{attribute 'Tc2GvlVarNames'}
VAR_GLOBAL

(* xxxxxxxxxxxxxxxxxxxxxxxxxxxxxxxx OUTPUT DWORD LINK with %MX10000-MX19000  xxxxxxxxxxxxxxxxxxxxxxxxxxxxxxxx*)
(*========================================================================*)

	WY10000 :DWORD; (* %MD10000 - GENERAL ALARM RESET IND (-100S1) *)
	WY10001 :DWORD; (* %MD10004 - GENERAL BUZZER RESET IND (-100S2) *)
	WY10002 :DWORD; (* %MD10008 - GENERAL BUZZER TONE 1 (-150H3) *)
	WY10003 :DWORD; (* %MD10012 - GENERAL BUZZER TONE 2 (-150H3) *)
	WY10004 :DWORD; (* %MD10016 - GENERAL TOWER LIGHT IND - RED (-150H5) *)
	WY10005 :DWORD; (* %MD10020 - GENERAL TOWER LIGHT IND - YELLOW (-150H5) *)
	WY10006 :DWORD; (* %MD10024 - GENERAL TOWER LIGHT IND - GREEN (-150H5) *)
	WY10007 :DWORD; (* %MD10028 - RESERVED *)
	WY10008 :DWORD; (* %MD10032 - RESERVED *)
	WY10009 :DWORD; (* %MD10036 - RESERVED *)
	WY10010 :DWORD; (* %MD10040 - RESERVED *)
	WY10011 :DWORD; (* %MD10044 - RESERVED *)
	WY10012 :DWORD; (* %MD10048 - RESERVED *)
	WY10013 :DWORD; (* %MD10052 - RESERVED *)
	WY10014 :DWORD; (* %MD10056 - RESERVED *)
	WY10015 :DWORD; (* %MD10060 - RESERVED *)

	WY10100 :DWORD; (* %MD10100 - STN 1 PROCESS TANK PUMP ON/OFF (-50K1) *)
	WY10101 :DWORD; (* %MD10104 - STN 2 PROCESS TANK PUMP ON/OFF (-51K1) *)
	WY10102 :DWORD; (* %MD10108 - STN 3 PROCESS TANK PUMP ON/OFF (-52K1) *)
	WY10103 :DWORD; (* %MD10112 - STN 5 VACUUM PUMP ON/OFF (-56K1) *)
	WY10104 :DWORD; (* %MD10116 - STN 2&3 AGITATION MOTOR ON/OFF (-25K1) *)
	WY10105 :DWORD; (* %MD10120 - STN 5 BLOWER ON/OFF (-65K1) *)
	WY10106 :DWORD; (* %MD10124 - STN 1 SUB PROCESS TANK STIRRING MOTOR ON/OFF (-26K1) *)
	WY10107 :DWORD; (* %MD10128 - DETERGENT TANK 1 STIRRING MOTOR ON/OFF (-27K1) *)
	WY10108 :DWORD; (* %MD10132 - STN 1 ULTRASONIC ON/OFF (-16K1) *)
	WY10109 :DWORD; (* %MD10136 - STN 2 ULTRASONIC ON/OFF (-17K1) *)
	WY10110 :DWORD; (* %MD10140 - STN 3 ULTRASONIC ON/OFF (-18K1) *)
	WY10111 :DWORD; (* %MD10144 - STN 1 ELECTRIC ACTUATOR ON/OFF (-21K1) *)
	WY10112 :DWORD; (* %MD10148 - STN 2 ELECTRIC ACTUATOR ON/OFF (-22K1) *)
	WY10113 :DWORD; (* %MD10152 - STN 3 ELECTRIC ACTUATOR ON/OFF (-23K1) *)
	WY10114 :DWORD; (* %MD10156 - RESERVED *)
	WY10115 :DWORD; (* %MD10160 - RESERVED *)

	WY10200 :DWORD; (* %MD10200 - STN 5 PROCESS TANK HEATER A ON/OFF (-70K1) *)
	WY10201 :DWORD; (* %MD10204 - STN 5 PROCESS TANK HEATER B ON/OFF (-71K1) *)
	WY10202 :DWORD; (* %MD10208 - STN 1 SUB PROCESS TANK HEATER ON/OFF (-72K1) *)
	WY10203 :DWORD; (* %MD10212 - STN 2 SUB PROCESS TANK HEATER ON/OFF (-73K1) *)
	WY10204 :DWORD; (* %MD10216 - STN 3 SUB PROCESS TANK HEATER ON/OFF (-74K1) *)
	WY10205 :DWORD; (* %MD10220 - MAIN INC HEATER ON/OFF   (-75K1) *)
	WY10206 :DWORD; (* %MD10224 - STN 1 ULTRASONIC FREQ ON/OFF (-16U1) *)
	WY10207 :DWORD; (* %MD10228 - STN 2 ULTRASONIC FREQ ON/OFF (-17U1) *)
	WY10208 :DWORD; (* %MD10232 - STN 3 ULTRASONIC FREQ ON/OFF (-18U1) *)
	WY10209 :DWORD; (* %MD10236 - RESERVED *)
	WY10210 :DWORD; (* %MD10240 - RESERVED *)
	WY10211 :DWORD; (* %MD10244 - RESERVED *)
	WY10212 :DWORD; (* %MD10248 - RESERVED *)
	WY10213 :DWORD; (* %MD10252 - RESERVED *)
	WY10214 :DWORD; (* %MD10256 - RESERVED *)
	WY10215 :DWORD; (* %MD10260 - RESERVED *)

	WY11500 :DWORD; (* %MD11500 - STN 1 SLIDING DOOR - OPEN (-160Y1) *)
	WY11501 :DWORD; (* %MD11504 - STN 1 SLIDING DOOR - CLOSE (-160Y2) *)
	WY11502 :DWORD; (* %MD11508 - STN 4 SLIDING DOOR - OPEN (-160Y3) *)
	WY11503 :DWORD; (* %MD11512 - STN 4 SLIDING DOOR - CLOSE (-160Y4) *)
	WY11504 :DWORD; (* %MD11516 - STN 5 SLIDING DOOR - OPEN (-160Y5) *)
	WY11505 :DWORD; (* %MD11520 - STN 5 SLIDING DOOR - CLOSE (-160Y6) *)
	WY11506 :DWORD; (* %MD11524 - STN 5 SLIDING DOOR - CLAMP (-160Y7) *)
	WY11507 :DWORD; (* %MD11528 - STN 5 SLIDING DOOR - UNCLAMP (-160Y8) *)
	WY11508 :DWORD; (* %MD11532 - LD CYLINDER - UP (-160Y9) *)
	WY11509 :DWORD; (* %MD11536 - LD CYLINDER - DOWN (-160Y10) *)
	WY11510 :DWORD; (* %MD11540 - LD CYLINDER - FRONT (-160Y11) *)
	WY11511 :DWORD; (* %MD11544 - LD CYLINDER - BACK (-160Y12) *)
	WY11512 :DWORD; (* %MD11548 - ULD CYLINDER - UP (-160Y13) *)
	WY11513 :DWORD; (* %MD11552 - ULD CYLINDER - DOWN (-160Y14) *)
	WY11514 :DWORD; (* %MD11556 - ULD CYLINDER - FRONT (-160Y15) *)
	WY11515 :DWORD; (* %MD11560 - ULD CYLINDER - BACK (-160Y16) *)

	WY11600 :DWORD; (* %MD11600 - GENERAL INCOMING DIW SUPPLY AVINC-1 (-161Y1) *)
	WY11601 :DWORD; (* %MD11604 - STN 1 PROCESS TANK INCOMING DI SUPPLY AV1-1 (-161Y2) *)
	WY11602 :DWORD; (* %MD11608 - STN 1 SUB TANK INCOMING DIW SUPPLY AV1-2 (-161Y3) *)
	WY11603 :DWORD; (* %MD11612 - STN 1 DETERGENT SUPPLY 3-2 WAY AV1-3 (-161Y4) *)
	WY11604 :DWORD; (* %MD11616 - STN 2 PROCESS TANK INCOMING DIW SUPPLY AV2-1 (-161Y5) *)
	WY11605 :DWORD; (* %MD11620 - STN 3 PROCESS TANK INCOMING DIW SUPPLY AV3-1 (-161Y6) *)
	WY11606 :DWORD; (* %MD11624 - STN 4 PROCESS TANK CDA DISCHARGE AV4-1 (-161Y7) *)
	WY11607 :DWORD; (* %MD11628 - STN 4 PROCESS TANK CDA DISCHARGE AV4-2 (-161Y8) *)
	WY11608 :DWORD; (* %MD11632 - STN 5 PROCESS TANK VACUUM SUCTION AV5-1 (-161Y9) *)
	WY11609 :DWORD; (* %MD11636 - STN 5 PROCESS TANK VACUUM RELEASE AV5-2 (-161Y10) *)
	WY11610 :DWORD; (* %MD11640 - STN 5 BLOWER PROTECTION BUTTLEFLY AV5-3 (-161Y11) *)
	WY11611 :DWORD; (* %MD11644 - STN 5 BLOWER PROTECTION BUTTLEFLY AV5-4 (-161Y12) *)
	WY11612 :DWORD; (* %MD11648 - FACILITY CHILL WATER SUPPLY AV5-5 (-161Y13) *)
	WY11613 :DWORD; (* %MD11652 - STN 4 & UNLOADING IONIZER CDA DISCHARGE AVION-1 (-161Y14,15) *)
	WY11614 :DWORD; (* %MD11656 - STN 4 IONIZER STATIC ELIMINATION STOP SIGNAL (-161U1) *)
	WY11615 :DWORD; (* %MD11660 - UNLOADING IONIZER STATIC ELIMINATION STOP SIGNAL (-161U2) *)

	WY11700 :DWORD; (* %MD11700 - STN 4 CDA CYLINDER - IN (-162Y1) *)
	WY11701 :DWORD; (* %MD11704 - STN 4 CDA CYLINDER - OUT (-162Y2) *)
	WY11702 :DWORD; (* %MD11708 - RAMP PUMP AV (-162Y3) *)
	WY11703 :DWORD; (* %MD11712 - RESERVED *)
	WY11704 :DWORD; (* %MD11716 - RESERVED *)
	WY11705 :DWORD; (* %MD11720 - RESERVED *)
	WY11706 :DWORD; (* %MD11724 - RESERVED *)
	WY11707 :DWORD; (* %MD11728 - RESERVED *)
	WY11708 :DWORD; (* %MD11732 - RESERVED *)
	WY11709 :DWORD; (* %MD11736 - RESERVED *)
	WY11710 :DWORD; (* %MD11740 - RESERVED *)
	WY11711 :DWORD; (* %MD11744 - RESERVED *)
	WY11712 :DWORD; (* %MD11748 - RESERVED *)
	WY11713 :DWORD; (* %MD11752 - RESERVED *)
	WY11714 :DWORD; (* %MD11756 - RESERVED *)
	WY11715 :DWORD; (* %MD11760 - RESERVED *)

(* xxxxxxxxxxxxxxxxxxxxxxxxxxxxxxxx OUTPUT BOOL LINK with %MX10000-MX19000  xxxxxxxxxxxxxxxxxxxxxxxxxxxxxxxx*)
(*========================================================================*)

	WY10000_00 AT  %MX10000.0 : BOOL; (*GENERAL ALARM RESET IND (-100S1) *)
	WY10000_01 AT  %MX10000.1 : BOOL; (*GENERAL ALARM RESET IND (-100S1) *)
	WY10000_02 AT  %MX10000.2 : BOOL; (*GENERAL ALARM RESET IND (-100S1) *)
	WY10000_03 AT  %MX10000.3 : BOOL; (*GENERAL ALARM RESET IND (-100S1) *)
	WY10000_04 AT  %MX10000.4 : BOOL; (*GENERAL ALARM RESET IND (-100S1) *)
	WY10000_05 AT  %MX10000.5 : BOOL; (*GENERAL ALARM RESET IND (-100S1) *)
	WY10000_06 AT  %MX10000.6 : BOOL; (*GENERAL ALARM RESET IND (-100S1) *)
	WY10000_07 AT  %MX10000.7 : BOOL; (*GENERAL ALARM RESET IND (-100S1) *)
	WY10000_08 AT  %MX10000.8 : BOOL; (*GENERAL ALARM RESET IND (-100S1) *)
	WY10000_09 AT  %MX10000.9 : BOOL; (*GENERAL ALARM RESET IND (-100S1) *)
	WY10000_10 AT  %MX10000.10 : BOOL; (*GENERAL ALARM RESET IND (-100S1) *)
	WY10000_11 AT  %MX10000.11 : BOOL; (*GENERAL ALARM RESET IND (-100S1) *)
	WY10000_12 AT  %MX10000.12 : BOOL; (*GENERAL ALARM RESET IND (-100S1) *)
	WY10000_13 AT  %MX10000.13 : BOOL; (*GENERAL ALARM RESET IND (-100S1) *)
	WY10000_14 AT  %MX10000.14 : BOOL; (*GENERAL ALARM RESET IND (-100S1) *)
	WY10000_15 AT  %MX10000.15 : BOOL; (*GENERAL ALARM RESET IND (-100S1) *)
	WY10000_16 AT  %MX10000.16 : BOOL; (*GENERAL ALARM RESET IND (-100S1) *)
	WY10000_17 AT  %MX10000.17 : BOOL; (*GENERAL ALARM RESET IND (-100S1) *)
	WY10000_18 AT  %MX10000.18 : BOOL; (*GENERAL ALARM RESET IND (-100S1) *)
	WY10000_19 AT  %MX10000.19 : BOOL; (*GENERAL ALARM RESET IND (-100S1) *)
	WY10000_20 AT  %MX10000.20 : BOOL; (*GENERAL ALARM RESET IND (-100S1) *)
	WY10000_21 AT  %MX10000.21 : BOOL; (*GENERAL ALARM RESET IND (-100S1) *)
	WY10000_22 AT  %MX10000.22 : BOOL; (*GENERAL ALARM RESET IND (-100S1) *)
	WY10000_23 AT  %MX10000.23 : BOOL; (*GENERAL ALARM RESET IND (-100S1) *)
	WY10000_24 AT  %MX10000.24 : BOOL; (*GENERAL ALARM RESET IND (-100S1) *)
	WY10000_25 AT  %MX10000.25 : BOOL; (*GENERAL ALARM RESET IND (-100S1) *)
	WY10000_26 AT  %MX10000.26 : BOOL; (*GENERAL ALARM RESET IND (-100S1) *)
	WY10000_27 AT  %MX10000.27 : BOOL; (*GENERAL ALARM RESET IND (-100S1) *)
	WY10000_28 AT  %MX10000.28 : BOOL; (*GENERAL ALARM RESET IND (-100S1) *)
	WY10000_29 AT  %MX10000.29 : BOOL; (*GENERAL ALARM RESET IND (-100S1) *)
	WY10000_30 AT  %MX10000.30 : BOOL; (*GENERAL ALARM RESET IND (-100S1) *)
	WY10000_31 AT  %MX10000.31 : BOOL; (*GENERAL ALARM RESET IND (-100S1) *)

	WY10001_00 AT  %MX10004.0 : BOOL; (*GENERAL BUZZER RESET IND (-100S2) *)
	WY10001_01 AT  %MX10004.1 : BOOL; (*GENERAL BUZZER RESET IND (-100S2) *)
	WY10001_02 AT  %MX10004.2 : BOOL; (*GENERAL BUZZER RESET IND (-100S2) *)
	WY10001_03 AT  %MX10004.3 : BOOL; (*GENERAL BUZZER RESET IND (-100S2) *)
	WY10001_04 AT  %MX10004.4 : BOOL; (*GENERAL BUZZER RESET IND (-100S2) *)
	WY10001_05 AT  %MX10004.5 : BOOL; (*GENERAL BUZZER RESET IND (-100S2) *)
	WY10001_06 AT  %MX10004.6 : BOOL; (*GENERAL BUZZER RESET IND (-100S2) *)
	WY10001_07 AT  %MX10004.7 : BOOL; (*GENERAL BUZZER RESET IND (-100S2) *)
	WY10001_08 AT  %MX10004.8 : BOOL; (*GENERAL BUZZER RESET IND (-100S2) *)
	WY10001_09 AT  %MX10004.9 : BOOL; (*GENERAL BUZZER RESET IND (-100S2) *)
	WY10001_10 AT  %MX10004.10 : BOOL; (*GENERAL BUZZER RESET IND (-100S2) *)
	WY10001_11 AT  %MX10004.11 : BOOL; (*GENERAL BUZZER RESET IND (-100S2) *)
	WY10001_12 AT  %MX10004.12 : BOOL; (*GENERAL BUZZER RESET IND (-100S2) *)
	WY10001_13 AT  %MX10004.13 : BOOL; (*GENERAL BUZZER RESET IND (-100S2) *)
	WY10001_14 AT  %MX10004.14 : BOOL; (*GENERAL BUZZER RESET IND (-100S2) *)
	WY10001_15 AT  %MX10004.15 : BOOL; (*GENERAL BUZZER RESET IND (-100S2) *)
	WY10001_16 AT  %MX10004.16 : BOOL; (*GENERAL BUZZER RESET IND (-100S2) *)
	WY10001_17 AT  %MX10004.17 : BOOL; (*GENERAL BUZZER RESET IND (-100S2) *)
	WY10001_18 AT  %MX10004.18 : BOOL; (*GENERAL BUZZER RESET IND (-100S2) *)
	WY10001_19 AT  %MX10004.19 : BOOL; (*GENERAL BUZZER RESET IND (-100S2) *)
	WY10001_20 AT  %MX10004.20 : BOOL; (*GENERAL BUZZER RESET IND (-100S2) *)
	WY10001_21 AT  %MX10004.21 : BOOL; (*GENERAL BUZZER RESET IND (-100S2) *)
	WY10001_22 AT  %MX10004.22 : BOOL; (*GENERAL BUZZER RESET IND (-100S2) *)
	WY10001_23 AT  %MX10004.23 : BOOL; (*GENERAL BUZZER RESET IND (-100S2) *)
	WY10001_24 AT  %MX10004.24 : BOOL; (*GENERAL BUZZER RESET IND (-100S2) *)
	WY10001_25 AT  %MX10004.25 : BOOL; (*GENERAL BUZZER RESET IND (-100S2) *)
	WY10001_26 AT  %MX10004.26 : BOOL; (*GENERAL BUZZER RESET IND (-100S2) *)
	WY10001_27 AT  %MX10004.27 : BOOL; (*GENERAL BUZZER RESET IND (-100S2) *)
	WY10001_28 AT  %MX10004.28 : BOOL; (*GENERAL BUZZER RESET IND (-100S2) *)
	WY10001_29 AT  %MX10004.29 : BOOL; (*GENERAL BUZZER RESET IND (-100S2) *)
	WY10001_30 AT  %MX10004.30 : BOOL; (*GENERAL BUZZER RESET IND (-100S2) *)
	WY10001_31 AT  %MX10004.31 : BOOL; (*GENERAL BUZZER RESET IND (-100S2) *)

	WY10002_00 AT  %MX10008.0 : BOOL; (*GENERAL BUZZER TONE 1 (-150H3) *)
	WY10002_01 AT  %MX10008.1 : BOOL; (*GENERAL BUZZER TONE 1 (-150H3) *)
	WY10002_02 AT  %MX10008.2 : BOOL; (*GENERAL BUZZER TONE 1 (-150H3) *)
	WY10002_03 AT  %MX10008.3 : BOOL; (*GENERAL BUZZER TONE 1 (-150H3) *)
	WY10002_04 AT  %MX10008.4 : BOOL; (*GENERAL BUZZER TONE 1 (-150H3) *)
	WY10002_05 AT  %MX10008.5 : BOOL; (*GENERAL BUZZER TONE 1 (-150H3) *)
	WY10002_06 AT  %MX10008.6 : BOOL; (*GENERAL BUZZER TONE 1 (-150H3) *)
	WY10002_07 AT  %MX10008.7 : BOOL; (*GENERAL BUZZER TONE 1 (-150H3) *)
	WY10002_08 AT  %MX10008.8 : BOOL; (*GENERAL BUZZER TONE 1 (-150H3) *)
	WY10002_09 AT  %MX10008.9 : BOOL; (*GENERAL BUZZER TONE 1 (-150H3) *)
	WY10002_10 AT  %MX10008.10 : BOOL; (*GENERAL BUZZER TONE 1 (-150H3) *)
	WY10002_11 AT  %MX10008.11 : BOOL; (*GENERAL BUZZER TONE 1 (-150H3) *)
	WY10002_12 AT  %MX10008.12 : BOOL; (*GENERAL BUZZER TONE 1 (-150H3) *)
	WY10002_13 AT  %MX10008.13 : BOOL; (*GENERAL BUZZER TONE 1 (-150H3) *)
	WY10002_14 AT  %MX10008.14 : BOOL; (*GENERAL BUZZER TONE 1 (-150H3) *)
	WY10002_15 AT  %MX10008.15 : BOOL; (*GENERAL BUZZER TONE 1 (-150H3) *)
	WY10002_16 AT  %MX10008.16 : BOOL; (*GENERAL BUZZER TONE 1 (-150H3) *)
	WY10002_17 AT  %MX10008.17 : BOOL; (*GENERAL BUZZER TONE 1 (-150H3) *)
	WY10002_18 AT  %MX10008.18 : BOOL; (*GENERAL BUZZER TONE 1 (-150H3) *)
	WY10002_19 AT  %MX10008.19 : BOOL; (*GENERAL BUZZER TONE 1 (-150H3) *)
	WY10002_20 AT  %MX10008.20 : BOOL; (*GENERAL BUZZER TONE 1 (-150H3) *)
	WY10002_21 AT  %MX10008.21 : BOOL; (*GENERAL BUZZER TONE 1 (-150H3) *)
	WY10002_22 AT  %MX10008.22 : BOOL; (*GENERAL BUZZER TONE 1 (-150H3) *)
	WY10002_23 AT  %MX10008.23 : BOOL; (*GENERAL BUZZER TONE 1 (-150H3) *)
	WY10002_24 AT  %MX10008.24 : BOOL; (*GENERAL BUZZER TONE 1 (-150H3) *)
	WY10002_25 AT  %MX10008.25 : BOOL; (*GENERAL BUZZER TONE 1 (-150H3) *)
	WY10002_26 AT  %MX10008.26 : BOOL; (*GENERAL BUZZER TONE 1 (-150H3) *)
	WY10002_27 AT  %MX10008.27 : BOOL; (*GENERAL BUZZER TONE 1 (-150H3) *)
	WY10002_28 AT  %MX10008.28 : BOOL; (*GENERAL BUZZER TONE 1 (-150H3) *)
	WY10002_29 AT  %MX10008.29 : BOOL; (*GENERAL BUZZER TONE 1 (-150H3) *)
	WY10002_30 AT  %MX10008.30 : BOOL; (*GENERAL BUZZER TONE 1 (-150H3) *)
	WY10002_31 AT  %MX10008.31 : BOOL; (*GENERAL BUZZER TONE 1 (-150H3) *)

	WY10003_00 AT  %MX10012.0 : BOOL; (*GENERAL BUZZER TONE 2 (-150H3) *)
	WY10003_01 AT  %MX10012.1 : BOOL; (*GENERAL BUZZER TONE 2 (-150H3) *)
	WY10003_02 AT  %MX10012.2 : BOOL; (*GENERAL BUZZER TONE 2 (-150H3) *)
	WY10003_03 AT  %MX10012.3 : BOOL; (*GENERAL BUZZER TONE 2 (-150H3) *)
	WY10003_04 AT  %MX10012.4 : BOOL; (*GENERAL BUZZER TONE 2 (-150H3) *)
	WY10003_05 AT  %MX10012.5 : BOOL; (*GENERAL BUZZER TONE 2 (-150H3) *)
	WY10003_06 AT  %MX10012.6 : BOOL; (*GENERAL BUZZER TONE 2 (-150H3) *)
	WY10003_07 AT  %MX10012.7 : BOOL; (*GENERAL BUZZER TONE 2 (-150H3) *)
	WY10003_08 AT  %MX10012.8 : BOOL; (*GENERAL BUZZER TONE 2 (-150H3) *)
	WY10003_09 AT  %MX10012.9 : BOOL; (*GENERAL BUZZER TONE 2 (-150H3) *)
	WY10003_10 AT  %MX10012.10 : BOOL; (*GENERAL BUZZER TONE 2 (-150H3) *)
	WY10003_11 AT  %MX10012.11 : BOOL; (*GENERAL BUZZER TONE 2 (-150H3) *)
	WY10003_12 AT  %MX10012.12 : BOOL; (*GENERAL BUZZER TONE 2 (-150H3) *)
	WY10003_13 AT  %MX10012.13 : BOOL; (*GENERAL BUZZER TONE 2 (-150H3) *)
	WY10003_14 AT  %MX10012.14 : BOOL; (*GENERAL BUZZER TONE 2 (-150H3) *)
	WY10003_15 AT  %MX10012.15 : BOOL; (*GENERAL BUZZER TONE 2 (-150H3) *)
	WY10003_16 AT  %MX10012.16 : BOOL; (*GENERAL BUZZER TONE 2 (-150H3) *)
	WY10003_17 AT  %MX10012.17 : BOOL; (*GENERAL BUZZER TONE 2 (-150H3) *)
	WY10003_18 AT  %MX10012.18 : BOOL; (*GENERAL BUZZER TONE 2 (-150H3) *)
	WY10003_19 AT  %MX10012.19 : BOOL; (*GENERAL BUZZER TONE 2 (-150H3) *)
	WY10003_20 AT  %MX10012.20 : BOOL; (*GENERAL BUZZER TONE 2 (-150H3) *)
	WY10003_21 AT  %MX10012.21 : BOOL; (*GENERAL BUZZER TONE 2 (-150H3) *)
	WY10003_22 AT  %MX10012.22 : BOOL; (*GENERAL BUZZER TONE 2 (-150H3) *)
	WY10003_23 AT  %MX10012.23 : BOOL; (*GENERAL BUZZER TONE 2 (-150H3) *)
	WY10003_24 AT  %MX10012.24 : BOOL; (*GENERAL BUZZER TONE 2 (-150H3) *)
	WY10003_25 AT  %MX10012.25 : BOOL; (*GENERAL BUZZER TONE 2 (-150H3) *)
	WY10003_26 AT  %MX10012.26 : BOOL; (*GENERAL BUZZER TONE 2 (-150H3) *)
	WY10003_27 AT  %MX10012.27 : BOOL; (*GENERAL BUZZER TONE 2 (-150H3) *)
	WY10003_28 AT  %MX10012.28 : BOOL; (*GENERAL BUZZER TONE 2 (-150H3) *)
	WY10003_29 AT  %MX10012.29 : BOOL; (*GENERAL BUZZER TONE 2 (-150H3) *)
	WY10003_30 AT  %MX10012.30 : BOOL; (*GENERAL BUZZER TONE 2 (-150H3) *)
	WY10003_31 AT  %MX10012.31 : BOOL; (*GENERAL BUZZER TONE 2 (-150H3) *)

	WY10004_00 AT  %MX10016.0 : BOOL; (*GENERAL TOWER LIGHT IND - RED (-150H5) *)
	WY10004_01 AT  %MX10016.1 : BOOL; (*GENERAL TOWER LIGHT IND - RED (-150H5) *)
	WY10004_02 AT  %MX10016.2 : BOOL; (*GENERAL TOWER LIGHT IND - RED (-150H5) *)
	WY10004_03 AT  %MX10016.3 : BOOL; (*GENERAL TOWER LIGHT IND - RED (-150H5) *)
	WY10004_04 AT  %MX10016.4 : BOOL; (*GENERAL TOWER LIGHT IND - RED (-150H5) *)
	WY10004_05 AT  %MX10016.5 : BOOL; (*GENERAL TOWER LIGHT IND - RED (-150H5) *)
	WY10004_06 AT  %MX10016.6 : BOOL; (*GENERAL TOWER LIGHT IND - RED (-150H5) *)
	WY10004_07 AT  %MX10016.7 : BOOL; (*GENERAL TOWER LIGHT IND - RED (-150H5) *)
	WY10004_08 AT  %MX10016.8 : BOOL; (*GENERAL TOWER LIGHT IND - RED (-150H5) *)
	WY10004_09 AT  %MX10016.9 : BOOL; (*GENERAL TOWER LIGHT IND - RED (-150H5) *)
	WY10004_10 AT  %MX10016.10 : BOOL; (*GENERAL TOWER LIGHT IND - RED (-150H5) *)
	WY10004_11 AT  %MX10016.11 : BOOL; (*GENERAL TOWER LIGHT IND - RED (-150H5) *)
	WY10004_12 AT  %MX10016.12 : BOOL; (*GENERAL TOWER LIGHT IND - RED (-150H5) *)
	WY10004_13 AT  %MX10016.13 : BOOL; (*GENERAL TOWER LIGHT IND - RED (-150H5) *)
	WY10004_14 AT  %MX10016.14 : BOOL; (*GENERAL TOWER LIGHT IND - RED (-150H5) *)
	WY10004_15 AT  %MX10016.15 : BOOL; (*GENERAL TOWER LIGHT IND - RED (-150H5) *)
	WY10004_16 AT  %MX10016.16 : BOOL; (*GENERAL TOWER LIGHT IND - RED (-150H5) *)
	WY10004_17 AT  %MX10016.17 : BOOL; (*GENERAL TOWER LIGHT IND - RED (-150H5) *)
	WY10004_18 AT  %MX10016.18 : BOOL; (*GENERAL TOWER LIGHT IND - RED (-150H5) *)
	WY10004_19 AT  %MX10016.19 : BOOL; (*GENERAL TOWER LIGHT IND - RED (-150H5) *)
	WY10004_20 AT  %MX10016.20 : BOOL; (*GENERAL TOWER LIGHT IND - RED (-150H5) *)
	WY10004_21 AT  %MX10016.21 : BOOL; (*GENERAL TOWER LIGHT IND - RED (-150H5) *)
	WY10004_22 AT  %MX10016.22 : BOOL; (*GENERAL TOWER LIGHT IND - RED (-150H5) *)
	WY10004_23 AT  %MX10016.23 : BOOL; (*GENERAL TOWER LIGHT IND - RED (-150H5) *)
	WY10004_24 AT  %MX10016.24 : BOOL; (*GENERAL TOWER LIGHT IND - RED (-150H5) *)
	WY10004_25 AT  %MX10016.25 : BOOL; (*GENERAL TOWER LIGHT IND - RED (-150H5) *)
	WY10004_26 AT  %MX10016.26 : BOOL; (*GENERAL TOWER LIGHT IND - RED (-150H5) *)
	WY10004_27 AT  %MX10016.27 : BOOL; (*GENERAL TOWER LIGHT IND - RED (-150H5) *)
	WY10004_28 AT  %MX10016.28 : BOOL; (*GENERAL TOWER LIGHT IND - RED (-150H5) *)
	WY10004_29 AT  %MX10016.29 : BOOL; (*GENERAL TOWER LIGHT IND - RED (-150H5) *)
	WY10004_30 AT  %MX10016.30 : BOOL; (*GENERAL TOWER LIGHT IND - RED (-150H5) *)
	WY10004_31 AT  %MX10016.31 : BOOL; (*GENERAL TOWER LIGHT IND - RED (-150H5) *)

	WY10005_00 AT  %MX10020.0 : BOOL; (*GENERAL TOWER LIGHT IND - YELLOW (-150H5) *)
	WY10005_01 AT  %MX10020.1 : BOOL; (*GENERAL TOWER LIGHT IND - YELLOW (-150H5) *)
	WY10005_02 AT  %MX10020.2 : BOOL; (*GENERAL TOWER LIGHT IND - YELLOW (-150H5) *)
	WY10005_03 AT  %MX10020.3 : BOOL; (*GENERAL TOWER LIGHT IND - YELLOW (-150H5) *)
	WY10005_04 AT  %MX10020.4 : BOOL; (*GENERAL TOWER LIGHT IND - YELLOW (-150H5) *)
	WY10005_05 AT  %MX10020.5 : BOOL; (*GENERAL TOWER LIGHT IND - YELLOW (-150H5) *)
	WY10005_06 AT  %MX10020.6 : BOOL; (*GENERAL TOWER LIGHT IND - YELLOW (-150H5) *)
	WY10005_07 AT  %MX10020.7 : BOOL; (*GENERAL TOWER LIGHT IND - YELLOW (-150H5) *)
	WY10005_08 AT  %MX10020.8 : BOOL; (*GENERAL TOWER LIGHT IND - YELLOW (-150H5) *)
	WY10005_09 AT  %MX10020.9 : BOOL; (*GENERAL TOWER LIGHT IND - YELLOW (-150H5) *)
	WY10005_10 AT  %MX10020.10 : BOOL; (*GENERAL TOWER LIGHT IND - YELLOW (-150H5) *)
	WY10005_11 AT  %MX10020.11 : BOOL; (*GENERAL TOWER LIGHT IND - YELLOW (-150H5) *)
	WY10005_12 AT  %MX10020.12 : BOOL; (*GENERAL TOWER LIGHT IND - YELLOW (-150H5) *)
	WY10005_13 AT  %MX10020.13 : BOOL; (*GENERAL TOWER LIGHT IND - YELLOW (-150H5) *)
	WY10005_14 AT  %MX10020.14 : BOOL; (*GENERAL TOWER LIGHT IND - YELLOW (-150H5) *)
	WY10005_15 AT  %MX10020.15 : BOOL; (*GENERAL TOWER LIGHT IND - YELLOW (-150H5) *)
	WY10005_16 AT  %MX10020.16 : BOOL; (*GENERAL TOWER LIGHT IND - YELLOW (-150H5) *)
	WY10005_17 AT  %MX10020.17 : BOOL; (*GENERAL TOWER LIGHT IND - YELLOW (-150H5) *)
	WY10005_18 AT  %MX10020.18 : BOOL; (*GENERAL TOWER LIGHT IND - YELLOW (-150H5) *)
	WY10005_19 AT  %MX10020.19 : BOOL; (*GENERAL TOWER LIGHT IND - YELLOW (-150H5) *)
	WY10005_20 AT  %MX10020.20 : BOOL; (*GENERAL TOWER LIGHT IND - YELLOW (-150H5) *)
	WY10005_21 AT  %MX10020.21 : BOOL; (*GENERAL TOWER LIGHT IND - YELLOW (-150H5) *)
	WY10005_22 AT  %MX10020.22 : BOOL; (*GENERAL TOWER LIGHT IND - YELLOW (-150H5) *)
	WY10005_23 AT  %MX10020.23 : BOOL; (*GENERAL TOWER LIGHT IND - YELLOW (-150H5) *)
	WY10005_24 AT  %MX10020.24 : BOOL; (*GENERAL TOWER LIGHT IND - YELLOW (-150H5) *)
	WY10005_25 AT  %MX10020.25 : BOOL; (*GENERAL TOWER LIGHT IND - YELLOW (-150H5) *)
	WY10005_26 AT  %MX10020.26 : BOOL; (*GENERAL TOWER LIGHT IND - YELLOW (-150H5) *)
	WY10005_27 AT  %MX10020.27 : BOOL; (*GENERAL TOWER LIGHT IND - YELLOW (-150H5) *)
	WY10005_28 AT  %MX10020.28 : BOOL; (*GENERAL TOWER LIGHT IND - YELLOW (-150H5) *)
	WY10005_29 AT  %MX10020.29 : BOOL; (*GENERAL TOWER LIGHT IND - YELLOW (-150H5) *)
	WY10005_30 AT  %MX10020.30 : BOOL; (*GENERAL TOWER LIGHT IND - YELLOW (-150H5) *)
	WY10005_31 AT  %MX10020.31 : BOOL; (*GENERAL TOWER LIGHT IND - YELLOW (-150H5) *)

	WY10006_00 AT  %MX10024.0 : BOOL; (*GENERAL TOWER LIGHT IND - GREEN (-150H5) *)
	WY10006_01 AT  %MX10024.1 : BOOL; (*GENERAL TOWER LIGHT IND - GREEN (-150H5) *)
	WY10006_02 AT  %MX10024.2 : BOOL; (*GENERAL TOWER LIGHT IND - GREEN (-150H5) *)
	WY10006_03 AT  %MX10024.3 : BOOL; (*GENERAL TOWER LIGHT IND - GREEN (-150H5) *)
	WY10006_04 AT  %MX10024.4 : BOOL; (*GENERAL TOWER LIGHT IND - GREEN (-150H5) *)
	WY10006_05 AT  %MX10024.5 : BOOL; (*GENERAL TOWER LIGHT IND - GREEN (-150H5) *)
	WY10006_06 AT  %MX10024.6 : BOOL; (*GENERAL TOWER LIGHT IND - GREEN (-150H5) *)
	WY10006_07 AT  %MX10024.7 : BOOL; (*GENERAL TOWER LIGHT IND - GREEN (-150H5) *)
	WY10006_08 AT  %MX10024.8 : BOOL; (*GENERAL TOWER LIGHT IND - GREEN (-150H5) *)
	WY10006_09 AT  %MX10024.9 : BOOL; (*GENERAL TOWER LIGHT IND - GREEN (-150H5) *)
	WY10006_10 AT  %MX10024.10 : BOOL; (*GENERAL TOWER LIGHT IND - GREEN (-150H5) *)
	WY10006_11 AT  %MX10024.11 : BOOL; (*GENERAL TOWER LIGHT IND - GREEN (-150H5) *)
	WY10006_12 AT  %MX10024.12 : BOOL; (*GENERAL TOWER LIGHT IND - GREEN (-150H5) *)
	WY10006_13 AT  %MX10024.13 : BOOL; (*GENERAL TOWER LIGHT IND - GREEN (-150H5) *)
	WY10006_14 AT  %MX10024.14 : BOOL; (*GENERAL TOWER LIGHT IND - GREEN (-150H5) *)
	WY10006_15 AT  %MX10024.15 : BOOL; (*GENERAL TOWER LIGHT IND - GREEN (-150H5) *)
	WY10006_16 AT  %MX10024.16 : BOOL; (*GENERAL TOWER LIGHT IND - GREEN (-150H5) *)
	WY10006_17 AT  %MX10024.17 : BOOL; (*GENERAL TOWER LIGHT IND - GREEN (-150H5) *)
	WY10006_18 AT  %MX10024.18 : BOOL; (*GENERAL TOWER LIGHT IND - GREEN (-150H5) *)
	WY10006_19 AT  %MX10024.19 : BOOL; (*GENERAL TOWER LIGHT IND - GREEN (-150H5) *)
	WY10006_20 AT  %MX10024.20 : BOOL; (*GENERAL TOWER LIGHT IND - GREEN (-150H5) *)
	WY10006_21 AT  %MX10024.21 : BOOL; (*GENERAL TOWER LIGHT IND - GREEN (-150H5) *)
	WY10006_22 AT  %MX10024.22 : BOOL; (*GENERAL TOWER LIGHT IND - GREEN (-150H5) *)
	WY10006_23 AT  %MX10024.23 : BOOL; (*GENERAL TOWER LIGHT IND - GREEN (-150H5) *)
	WY10006_24 AT  %MX10024.24 : BOOL; (*GENERAL TOWER LIGHT IND - GREEN (-150H5) *)
	WY10006_25 AT  %MX10024.25 : BOOL; (*GENERAL TOWER LIGHT IND - GREEN (-150H5) *)
	WY10006_26 AT  %MX10024.26 : BOOL; (*GENERAL TOWER LIGHT IND - GREEN (-150H5) *)
	WY10006_27 AT  %MX10024.27 : BOOL; (*GENERAL TOWER LIGHT IND - GREEN (-150H5) *)
	WY10006_28 AT  %MX10024.28 : BOOL; (*GENERAL TOWER LIGHT IND - GREEN (-150H5) *)
	WY10006_29 AT  %MX10024.29 : BOOL; (*GENERAL TOWER LIGHT IND - GREEN (-150H5) *)
	WY10006_30 AT  %MX10024.30 : BOOL; (*GENERAL TOWER LIGHT IND - GREEN (-150H5) *)
	WY10006_31 AT  %MX10024.31 : BOOL; (*GENERAL TOWER LIGHT IND - GREEN (-150H5) *)

	WY10007_00 AT  %MX10028.0 : BOOL; (*RESERVED *)
	WY10007_01 AT  %MX10028.1 : BOOL; (*RESERVED *)
	WY10007_02 AT  %MX10028.2 : BOOL; (*RESERVED *)
	WY10007_03 AT  %MX10028.3 : BOOL; (*RESERVED *)
	WY10007_04 AT  %MX10028.4 : BOOL; (*RESERVED *)
	WY10007_05 AT  %MX10028.5 : BOOL; (*RESERVED *)
	WY10007_06 AT  %MX10028.6 : BOOL; (*RESERVED *)
	WY10007_07 AT  %MX10028.7 : BOOL; (*RESERVED *)
	WY10007_08 AT  %MX10028.8 : BOOL; (*RESERVED *)
	WY10007_09 AT  %MX10028.9 : BOOL; (*RESERVED *)
	WY10007_10 AT  %MX10028.10 : BOOL; (*RESERVED *)
	WY10007_11 AT  %MX10028.11 : BOOL; (*RESERVED *)
	WY10007_12 AT  %MX10028.12 : BOOL; (*RESERVED *)
	WY10007_13 AT  %MX10028.13 : BOOL; (*RESERVED *)
	WY10007_14 AT  %MX10028.14 : BOOL; (*RESERVED *)
	WY10007_15 AT  %MX10028.15 : BOOL; (*RESERVED *)
	WY10007_16 AT  %MX10028.16 : BOOL; (*RESERVED *)
	WY10007_17 AT  %MX10028.17 : BOOL; (*RESERVED *)
	WY10007_18 AT  %MX10028.18 : BOOL; (*RESERVED *)
	WY10007_19 AT  %MX10028.19 : BOOL; (*RESERVED *)
	WY10007_20 AT  %MX10028.20 : BOOL; (*RESERVED *)
	WY10007_21 AT  %MX10028.21 : BOOL; (*RESERVED *)
	WY10007_22 AT  %MX10028.22 : BOOL; (*RESERVED *)
	WY10007_23 AT  %MX10028.23 : BOOL; (*RESERVED *)
	WY10007_24 AT  %MX10028.24 : BOOL; (*RESERVED *)
	WY10007_25 AT  %MX10028.25 : BOOL; (*RESERVED *)
	WY10007_26 AT  %MX10028.26 : BOOL; (*RESERVED *)
	WY10007_27 AT  %MX10028.27 : BOOL; (*RESERVED *)
	WY10007_28 AT  %MX10028.28 : BOOL; (*RESERVED *)
	WY10007_29 AT  %MX10028.29 : BOOL; (*RESERVED *)
	WY10007_30 AT  %MX10028.30 : BOOL; (*RESERVED *)
	WY10007_31 AT  %MX10028.31 : BOOL; (*RESERVED *)

	WY10008_00 AT  %MX10032.0 : BOOL; (*RESERVED *)
	WY10008_01 AT  %MX10032.1 : BOOL; (*RESERVED *)
	WY10008_02 AT  %MX10032.2 : BOOL; (*RESERVED *)
	WY10008_03 AT  %MX10032.3 : BOOL; (*RESERVED *)
	WY10008_04 AT  %MX10032.4 : BOOL; (*RESERVED *)
	WY10008_05 AT  %MX10032.5 : BOOL; (*RESERVED *)
	WY10008_06 AT  %MX10032.6 : BOOL; (*RESERVED *)
	WY10008_07 AT  %MX10032.7 : BOOL; (*RESERVED *)
	WY10008_08 AT  %MX10032.8 : BOOL; (*RESERVED *)
	WY10008_09 AT  %MX10032.9 : BOOL; (*RESERVED *)
	WY10008_10 AT  %MX10032.10 : BOOL; (*RESERVED *)
	WY10008_11 AT  %MX10032.11 : BOOL; (*RESERVED *)
	WY10008_12 AT  %MX10032.12 : BOOL; (*RESERVED *)
	WY10008_13 AT  %MX10032.13 : BOOL; (*RESERVED *)
	WY10008_14 AT  %MX10032.14 : BOOL; (*RESERVED *)
	WY10008_15 AT  %MX10032.15 : BOOL; (*RESERVED *)
	WY10008_16 AT  %MX10032.16 : BOOL; (*RESERVED *)
	WY10008_17 AT  %MX10032.17 : BOOL; (*RESERVED *)
	WY10008_18 AT  %MX10032.18 : BOOL; (*RESERVED *)
	WY10008_19 AT  %MX10032.19 : BOOL; (*RESERVED *)
	WY10008_20 AT  %MX10032.20 : BOOL; (*RESERVED *)
	WY10008_21 AT  %MX10032.21 : BOOL; (*RESERVED *)
	WY10008_22 AT  %MX10032.22 : BOOL; (*RESERVED *)
	WY10008_23 AT  %MX10032.23 : BOOL; (*RESERVED *)
	WY10008_24 AT  %MX10032.24 : BOOL; (*RESERVED *)
	WY10008_25 AT  %MX10032.25 : BOOL; (*RESERVED *)
	WY10008_26 AT  %MX10032.26 : BOOL; (*RESERVED *)
	WY10008_27 AT  %MX10032.27 : BOOL; (*RESERVED *)
	WY10008_28 AT  %MX10032.28 : BOOL; (*RESERVED *)
	WY10008_29 AT  %MX10032.29 : BOOL; (*RESERVED *)
	WY10008_30 AT  %MX10032.30 : BOOL; (*RESERVED *)
	WY10008_31 AT  %MX10032.31 : BOOL; (*RESERVED *)

	WY10009_00 AT  %MX10036.0 : BOOL; (*RESERVED *)
	WY10009_01 AT  %MX10036.1 : BOOL; (*RESERVED *)
	WY10009_02 AT  %MX10036.2 : BOOL; (*RESERVED *)
	WY10009_03 AT  %MX10036.3 : BOOL; (*RESERVED *)
	WY10009_04 AT  %MX10036.4 : BOOL; (*RESERVED *)
	WY10009_05 AT  %MX10036.5 : BOOL; (*RESERVED *)
	WY10009_06 AT  %MX10036.6 : BOOL; (*RESERVED *)
	WY10009_07 AT  %MX10036.7 : BOOL; (*RESERVED *)
	WY10009_08 AT  %MX10036.8 : BOOL; (*RESERVED *)
	WY10009_09 AT  %MX10036.9 : BOOL; (*RESERVED *)
	WY10009_10 AT  %MX10036.10 : BOOL; (*RESERVED *)
	WY10009_11 AT  %MX10036.11 : BOOL; (*RESERVED *)
	WY10009_12 AT  %MX10036.12 : BOOL; (*RESERVED *)
	WY10009_13 AT  %MX10036.13 : BOOL; (*RESERVED *)
	WY10009_14 AT  %MX10036.14 : BOOL; (*RESERVED *)
	WY10009_15 AT  %MX10036.15 : BOOL; (*RESERVED *)
	WY10009_16 AT  %MX10036.16 : BOOL; (*RESERVED *)
	WY10009_17 AT  %MX10036.17 : BOOL; (*RESERVED *)
	WY10009_18 AT  %MX10036.18 : BOOL; (*RESERVED *)
	WY10009_19 AT  %MX10036.19 : BOOL; (*RESERVED *)
	WY10009_20 AT  %MX10036.20 : BOOL; (*RESERVED *)
	WY10009_21 AT  %MX10036.21 : BOOL; (*RESERVED *)
	WY10009_22 AT  %MX10036.22 : BOOL; (*RESERVED *)
	WY10009_23 AT  %MX10036.23 : BOOL; (*RESERVED *)
	WY10009_24 AT  %MX10036.24 : BOOL; (*RESERVED *)
	WY10009_25 AT  %MX10036.25 : BOOL; (*RESERVED *)
	WY10009_26 AT  %MX10036.26 : BOOL; (*RESERVED *)
	WY10009_27 AT  %MX10036.27 : BOOL; (*RESERVED *)
	WY10009_28 AT  %MX10036.28 : BOOL; (*RESERVED *)
	WY10009_29 AT  %MX10036.29 : BOOL; (*RESERVED *)
	WY10009_30 AT  %MX10036.30 : BOOL; (*RESERVED *)
	WY10009_31 AT  %MX10036.31 : BOOL; (*RESERVED *)

	WY10010_00 AT  %MX10040.0 : BOOL; (*RESERVED *)
	WY10010_01 AT  %MX10040.1 : BOOL; (*RESERVED *)
	WY10010_02 AT  %MX10040.2 : BOOL; (*RESERVED *)
	WY10010_03 AT  %MX10040.3 : BOOL; (*RESERVED *)
	WY10010_04 AT  %MX10040.4 : BOOL; (*RESERVED *)
	WY10010_05 AT  %MX10040.5 : BOOL; (*RESERVED *)
	WY10010_06 AT  %MX10040.6 : BOOL; (*RESERVED *)
	WY10010_07 AT  %MX10040.7 : BOOL; (*RESERVED *)
	WY10010_08 AT  %MX10040.8 : BOOL; (*RESERVED *)
	WY10010_09 AT  %MX10040.9 : BOOL; (*RESERVED *)
	WY10010_10 AT  %MX10040.10 : BOOL; (*RESERVED *)
	WY10010_11 AT  %MX10040.11 : BOOL; (*RESERVED *)
	WY10010_12 AT  %MX10040.12 : BOOL; (*RESERVED *)
	WY10010_13 AT  %MX10040.13 : BOOL; (*RESERVED *)
	WY10010_14 AT  %MX10040.14 : BOOL; (*RESERVED *)
	WY10010_15 AT  %MX10040.15 : BOOL; (*RESERVED *)
	WY10010_16 AT  %MX10040.16 : BOOL; (*RESERVED *)
	WY10010_17 AT  %MX10040.17 : BOOL; (*RESERVED *)
	WY10010_18 AT  %MX10040.18 : BOOL; (*RESERVED *)
	WY10010_19 AT  %MX10040.19 : BOOL; (*RESERVED *)
	WY10010_20 AT  %MX10040.20 : BOOL; (*RESERVED *)
	WY10010_21 AT  %MX10040.21 : BOOL; (*RESERVED *)
	WY10010_22 AT  %MX10040.22 : BOOL; (*RESERVED *)
	WY10010_23 AT  %MX10040.23 : BOOL; (*RESERVED *)
	WY10010_24 AT  %MX10040.24 : BOOL; (*RESERVED *)
	WY10010_25 AT  %MX10040.25 : BOOL; (*RESERVED *)
	WY10010_26 AT  %MX10040.26 : BOOL; (*RESERVED *)
	WY10010_27 AT  %MX10040.27 : BOOL; (*RESERVED *)
	WY10010_28 AT  %MX10040.28 : BOOL; (*RESERVED *)
	WY10010_29 AT  %MX10040.29 : BOOL; (*RESERVED *)
	WY10010_30 AT  %MX10040.30 : BOOL; (*RESERVED *)
	WY10010_31 AT  %MX10040.31 : BOOL; (*RESERVED *)

	WY10011_00 AT  %MX10044.0 : BOOL; (*RESERVED *)
	WY10011_01 AT  %MX10044.1 : BOOL; (*RESERVED *)
	WY10011_02 AT  %MX10044.2 : BOOL; (*RESERVED *)
	WY10011_03 AT  %MX10044.3 : BOOL; (*RESERVED *)
	WY10011_04 AT  %MX10044.4 : BOOL; (*RESERVED *)
	WY10011_05 AT  %MX10044.5 : BOOL; (*RESERVED *)
	WY10011_06 AT  %MX10044.6 : BOOL; (*RESERVED *)
	WY10011_07 AT  %MX10044.7 : BOOL; (*RESERVED *)
	WY10011_08 AT  %MX10044.8 : BOOL; (*RESERVED *)
	WY10011_09 AT  %MX10044.9 : BOOL; (*RESERVED *)
	WY10011_10 AT  %MX10044.10 : BOOL; (*RESERVED *)
	WY10011_11 AT  %MX10044.11 : BOOL; (*RESERVED *)
	WY10011_12 AT  %MX10044.12 : BOOL; (*RESERVED *)
	WY10011_13 AT  %MX10044.13 : BOOL; (*RESERVED *)
	WY10011_14 AT  %MX10044.14 : BOOL; (*RESERVED *)
	WY10011_15 AT  %MX10044.15 : BOOL; (*RESERVED *)
	WY10011_16 AT  %MX10044.16 : BOOL; (*RESERVED *)
	WY10011_17 AT  %MX10044.17 : BOOL; (*RESERVED *)
	WY10011_18 AT  %MX10044.18 : BOOL; (*RESERVED *)
	WY10011_19 AT  %MX10044.19 : BOOL; (*RESERVED *)
	WY10011_20 AT  %MX10044.20 : BOOL; (*RESERVED *)
	WY10011_21 AT  %MX10044.21 : BOOL; (*RESERVED *)
	WY10011_22 AT  %MX10044.22 : BOOL; (*RESERVED *)
	WY10011_23 AT  %MX10044.23 : BOOL; (*RESERVED *)
	WY10011_24 AT  %MX10044.24 : BOOL; (*RESERVED *)
	WY10011_25 AT  %MX10044.25 : BOOL; (*RESERVED *)
	WY10011_26 AT  %MX10044.26 : BOOL; (*RESERVED *)
	WY10011_27 AT  %MX10044.27 : BOOL; (*RESERVED *)
	WY10011_28 AT  %MX10044.28 : BOOL; (*RESERVED *)
	WY10011_29 AT  %MX10044.29 : BOOL; (*RESERVED *)
	WY10011_30 AT  %MX10044.30 : BOOL; (*RESERVED *)
	WY10011_31 AT  %MX10044.31 : BOOL; (*RESERVED *)

	WY10012_00 AT  %MX10048.0 : BOOL; (*RESERVED *)
	WY10012_01 AT  %MX10048.1 : BOOL; (*RESERVED *)
	WY10012_02 AT  %MX10048.2 : BOOL; (*RESERVED *)
	WY10012_03 AT  %MX10048.3 : BOOL; (*RESERVED *)
	WY10012_04 AT  %MX10048.4 : BOOL; (*RESERVED *)
	WY10012_05 AT  %MX10048.5 : BOOL; (*RESERVED *)
	WY10012_06 AT  %MX10048.6 : BOOL; (*RESERVED *)
	WY10012_07 AT  %MX10048.7 : BOOL; (*RESERVED *)
	WY10012_08 AT  %MX10048.8 : BOOL; (*RESERVED *)
	WY10012_09 AT  %MX10048.9 : BOOL; (*RESERVED *)
	WY10012_10 AT  %MX10048.10 : BOOL; (*RESERVED *)
	WY10012_11 AT  %MX10048.11 : BOOL; (*RESERVED *)
	WY10012_12 AT  %MX10048.12 : BOOL; (*RESERVED *)
	WY10012_13 AT  %MX10048.13 : BOOL; (*RESERVED *)
	WY10012_14 AT  %MX10048.14 : BOOL; (*RESERVED *)
	WY10012_15 AT  %MX10048.15 : BOOL; (*RESERVED *)
	WY10012_16 AT  %MX10048.16 : BOOL; (*RESERVED *)
	WY10012_17 AT  %MX10048.17 : BOOL; (*RESERVED *)
	WY10012_18 AT  %MX10048.18 : BOOL; (*RESERVED *)
	WY10012_19 AT  %MX10048.19 : BOOL; (*RESERVED *)
	WY10012_20 AT  %MX10048.20 : BOOL; (*RESERVED *)
	WY10012_21 AT  %MX10048.21 : BOOL; (*RESERVED *)
	WY10012_22 AT  %MX10048.22 : BOOL; (*RESERVED *)
	WY10012_23 AT  %MX10048.23 : BOOL; (*RESERVED *)
	WY10012_24 AT  %MX10048.24 : BOOL; (*RESERVED *)
	WY10012_25 AT  %MX10048.25 : BOOL; (*RESERVED *)
	WY10012_26 AT  %MX10048.26 : BOOL; (*RESERVED *)
	WY10012_27 AT  %MX10048.27 : BOOL; (*RESERVED *)
	WY10012_28 AT  %MX10048.28 : BOOL; (*RESERVED *)
	WY10012_29 AT  %MX10048.29 : BOOL; (*RESERVED *)
	WY10012_30 AT  %MX10048.30 : BOOL; (*RESERVED *)
	WY10012_31 AT  %MX10048.31 : BOOL; (*RESERVED *)

	WY10013_00 AT  %MX10052.0 : BOOL; (*RESERVED *)
	WY10013_01 AT  %MX10052.1 : BOOL; (*RESERVED *)
	WY10013_02 AT  %MX10052.2 : BOOL; (*RESERVED *)
	WY10013_03 AT  %MX10052.3 : BOOL; (*RESERVED *)
	WY10013_04 AT  %MX10052.4 : BOOL; (*RESERVED *)
	WY10013_05 AT  %MX10052.5 : BOOL; (*RESERVED *)
	WY10013_06 AT  %MX10052.6 : BOOL; (*RESERVED *)
	WY10013_07 AT  %MX10052.7 : BOOL; (*RESERVED *)
	WY10013_08 AT  %MX10052.8 : BOOL; (*RESERVED *)
	WY10013_09 AT  %MX10052.9 : BOOL; (*RESERVED *)
	WY10013_10 AT  %MX10052.10 : BOOL; (*RESERVED *)
	WY10013_11 AT  %MX10052.11 : BOOL; (*RESERVED *)
	WY10013_12 AT  %MX10052.12 : BOOL; (*RESERVED *)
	WY10013_13 AT  %MX10052.13 : BOOL; (*RESERVED *)
	WY10013_14 AT  %MX10052.14 : BOOL; (*RESERVED *)
	WY10013_15 AT  %MX10052.15 : BOOL; (*RESERVED *)
	WY10013_16 AT  %MX10052.16 : BOOL; (*RESERVED *)
	WY10013_17 AT  %MX10052.17 : BOOL; (*RESERVED *)
	WY10013_18 AT  %MX10052.18 : BOOL; (*RESERVED *)
	WY10013_19 AT  %MX10052.19 : BOOL; (*RESERVED *)
	WY10013_20 AT  %MX10052.20 : BOOL; (*RESERVED *)
	WY10013_21 AT  %MX10052.21 : BOOL; (*RESERVED *)
	WY10013_22 AT  %MX10052.22 : BOOL; (*RESERVED *)
	WY10013_23 AT  %MX10052.23 : BOOL; (*RESERVED *)
	WY10013_24 AT  %MX10052.24 : BOOL; (*RESERVED *)
	WY10013_25 AT  %MX10052.25 : BOOL; (*RESERVED *)
	WY10013_26 AT  %MX10052.26 : BOOL; (*RESERVED *)
	WY10013_27 AT  %MX10052.27 : BOOL; (*RESERVED *)
	WY10013_28 AT  %MX10052.28 : BOOL; (*RESERVED *)
	WY10013_29 AT  %MX10052.29 : BOOL; (*RESERVED *)
	WY10013_30 AT  %MX10052.30 : BOOL; (*RESERVED *)
	WY10013_31 AT  %MX10052.31 : BOOL; (*RESERVED *)

	WY10014_00 AT  %MX10056.0 : BOOL; (*RESERVED *)
	WY10014_01 AT  %MX10056.1 : BOOL; (*RESERVED *)
	WY10014_02 AT  %MX10056.2 : BOOL; (*RESERVED *)
	WY10014_03 AT  %MX10056.3 : BOOL; (*RESERVED *)
	WY10014_04 AT  %MX10056.4 : BOOL; (*RESERVED *)
	WY10014_05 AT  %MX10056.5 : BOOL; (*RESERVED *)
	WY10014_06 AT  %MX10056.6 : BOOL; (*RESERVED *)
	WY10014_07 AT  %MX10056.7 : BOOL; (*RESERVED *)
	WY10014_08 AT  %MX10056.8 : BOOL; (*RESERVED *)
	WY10014_09 AT  %MX10056.9 : BOOL; (*RESERVED *)
	WY10014_10 AT  %MX10056.10 : BOOL; (*RESERVED *)
	WY10014_11 AT  %MX10056.11 : BOOL; (*RESERVED *)
	WY10014_12 AT  %MX10056.12 : BOOL; (*RESERVED *)
	WY10014_13 AT  %MX10056.13 : BOOL; (*RESERVED *)
	WY10014_14 AT  %MX10056.14 : BOOL; (*RESERVED *)
	WY10014_15 AT  %MX10056.15 : BOOL; (*RESERVED *)
	WY10014_16 AT  %MX10056.16 : BOOL; (*RESERVED *)
	WY10014_17 AT  %MX10056.17 : BOOL; (*RESERVED *)
	WY10014_18 AT  %MX10056.18 : BOOL; (*RESERVED *)
	WY10014_19 AT  %MX10056.19 : BOOL; (*RESERVED *)
	WY10014_20 AT  %MX10056.20 : BOOL; (*RESERVED *)
	WY10014_21 AT  %MX10056.21 : BOOL; (*RESERVED *)
	WY10014_22 AT  %MX10056.22 : BOOL; (*RESERVED *)
	WY10014_23 AT  %MX10056.23 : BOOL; (*RESERVED *)
	WY10014_24 AT  %MX10056.24 : BOOL; (*RESERVED *)
	WY10014_25 AT  %MX10056.25 : BOOL; (*RESERVED *)
	WY10014_26 AT  %MX10056.26 : BOOL; (*RESERVED *)
	WY10014_27 AT  %MX10056.27 : BOOL; (*RESERVED *)
	WY10014_28 AT  %MX10056.28 : BOOL; (*RESERVED *)
	WY10014_29 AT  %MX10056.29 : BOOL; (*RESERVED *)
	WY10014_30 AT  %MX10056.30 : BOOL; (*RESERVED *)
	WY10014_31 AT  %MX10056.31 : BOOL; (*RESERVED *)

	WY10015_00 AT  %MX10060.0 : BOOL; (*RESERVED *)
	WY10015_01 AT  %MX10060.1 : BOOL; (*RESERVED *)
	WY10015_02 AT  %MX10060.2 : BOOL; (*RESERVED *)
	WY10015_03 AT  %MX10060.3 : BOOL; (*RESERVED *)
	WY10015_04 AT  %MX10060.4 : BOOL; (*RESERVED *)
	WY10015_05 AT  %MX10060.5 : BOOL; (*RESERVED *)
	WY10015_06 AT  %MX10060.6 : BOOL; (*RESERVED *)
	WY10015_07 AT  %MX10060.7 : BOOL; (*RESERVED *)
	WY10015_08 AT  %MX10060.8 : BOOL; (*RESERVED *)
	WY10015_09 AT  %MX10060.9 : BOOL; (*RESERVED *)
	WY10015_10 AT  %MX10060.10 : BOOL; (*RESERVED *)
	WY10015_11 AT  %MX10060.11 : BOOL; (*RESERVED *)
	WY10015_12 AT  %MX10060.12 : BOOL; (*RESERVED *)
	WY10015_13 AT  %MX10060.13 : BOOL; (*RESERVED *)
	WY10015_14 AT  %MX10060.14 : BOOL; (*RESERVED *)
	WY10015_15 AT  %MX10060.15 : BOOL; (*RESERVED *)
	WY10015_16 AT  %MX10060.16 : BOOL; (*RESERVED *)
	WY10015_17 AT  %MX10060.17 : BOOL; (*RESERVED *)
	WY10015_18 AT  %MX10060.18 : BOOL; (*RESERVED *)
	WY10015_19 AT  %MX10060.19 : BOOL; (*RESERVED *)
	WY10015_20 AT  %MX10060.20 : BOOL; (*RESERVED *)
	WY10015_21 AT  %MX10060.21 : BOOL; (*RESERVED *)
	WY10015_22 AT  %MX10060.22 : BOOL; (*RESERVED *)
	WY10015_23 AT  %MX10060.23 : BOOL; (*RESERVED *)
	WY10015_24 AT  %MX10060.24 : BOOL; (*RESERVED *)
	WY10015_25 AT  %MX10060.25 : BOOL; (*RESERVED *)
	WY10015_26 AT  %MX10060.26 : BOOL; (*RESERVED *)
	WY10015_27 AT  %MX10060.27 : BOOL; (*RESERVED *)
	WY10015_28 AT  %MX10060.28 : BOOL; (*RESERVED *)
	WY10015_29 AT  %MX10060.29 : BOOL; (*RESERVED *)
	WY10015_30 AT  %MX10060.30 : BOOL; (*RESERVED *)
	WY10015_31 AT  %MX10060.31 : BOOL; (*RESERVED *)

	WY10100_00 AT  %MX10100.0 : BOOL; (*STN 1 PROCESS TANK PUMP ON/OFF (-50K1) *)
	WY10100_01 AT  %MX10100.1 : BOOL; (*STN 1 PROCESS TANK PUMP ON/OFF (-50K1) *)
	WY10100_02 AT  %MX10100.2 : BOOL; (*STN 1 PROCESS TANK PUMP ON/OFF (-50K1) *)
	WY10100_03 AT  %MX10100.3 : BOOL; (*STN 1 PROCESS TANK PUMP ON/OFF (-50K1) *)
	WY10100_04 AT  %MX10100.4 : BOOL; (*STN 1 PROCESS TANK PUMP ON/OFF (-50K1) *)
	WY10100_05 AT  %MX10100.5 : BOOL; (*STN 1 PROCESS TANK PUMP ON/OFF (-50K1) *)
	WY10100_06 AT  %MX10100.6 : BOOL; (*STN 1 PROCESS TANK PUMP ON/OFF (-50K1) *)
	WY10100_07 AT  %MX10100.7 : BOOL; (*STN 1 PROCESS TANK PUMP ON/OFF (-50K1) *)
	WY10100_08 AT  %MX10100.8 : BOOL; (*STN 1 PROCESS TANK PUMP ON/OFF (-50K1) *)
	WY10100_09 AT  %MX10100.9 : BOOL; (*STN 1 PROCESS TANK PUMP ON/OFF (-50K1) *)
	WY10100_10 AT  %MX10100.10 : BOOL; (*STN 1 PROCESS TANK PUMP ON/OFF (-50K1) *)
	WY10100_11 AT  %MX10100.11 : BOOL; (*STN 1 PROCESS TANK PUMP ON/OFF (-50K1) *)
	WY10100_12 AT  %MX10100.12 : BOOL; (*STN 1 PROCESS TANK PUMP ON/OFF (-50K1) *)
	WY10100_13 AT  %MX10100.13 : BOOL; (*STN 1 PROCESS TANK PUMP ON/OFF (-50K1) *)
	WY10100_14 AT  %MX10100.14 : BOOL; (*STN 1 PROCESS TANK PUMP ON/OFF (-50K1) *)
	WY10100_15 AT  %MX10100.15 : BOOL; (*STN 1 PROCESS TANK PUMP ON/OFF (-50K1) *)
	WY10100_16 AT  %MX10100.16 : BOOL; (*STN 1 PROCESS TANK PUMP ON/OFF (-50K1) *)
	WY10100_17 AT  %MX10100.17 : BOOL; (*STN 1 PROCESS TANK PUMP ON/OFF (-50K1) *)
	WY10100_18 AT  %MX10100.18 : BOOL; (*STN 1 PROCESS TANK PUMP ON/OFF (-50K1) *)
	WY10100_19 AT  %MX10100.19 : BOOL; (*STN 1 PROCESS TANK PUMP ON/OFF (-50K1) *)
	WY10100_20 AT  %MX10100.20 : BOOL; (*STN 1 PROCESS TANK PUMP ON/OFF (-50K1) *)
	WY10100_21 AT  %MX10100.21 : BOOL; (*STN 1 PROCESS TANK PUMP ON/OFF (-50K1) *)
	WY10100_22 AT  %MX10100.22 : BOOL; (*STN 1 PROCESS TANK PUMP ON/OFF (-50K1) *)
	WY10100_23 AT  %MX10100.23 : BOOL; (*STN 1 PROCESS TANK PUMP ON/OFF (-50K1) *)
	WY10100_24 AT  %MX10100.24 : BOOL; (*STN 1 PROCESS TANK PUMP ON/OFF (-50K1) *)
	WY10100_25 AT  %MX10100.25 : BOOL; (*STN 1 PROCESS TANK PUMP ON/OFF (-50K1) *)
	WY10100_26 AT  %MX10100.26 : BOOL; (*STN 1 PROCESS TANK PUMP ON/OFF (-50K1) *)
	WY10100_27 AT  %MX10100.27 : BOOL; (*STN 1 PROCESS TANK PUMP ON/OFF (-50K1) *)
	WY10100_28 AT  %MX10100.28 : BOOL; (*STN 1 PROCESS TANK PUMP ON/OFF (-50K1) *)
	WY10100_29 AT  %MX10100.29 : BOOL; (*STN 1 PROCESS TANK PUMP ON/OFF (-50K1) *)
	WY10100_30 AT  %MX10100.30 : BOOL; (*STN 1 PROCESS TANK PUMP ON/OFF (-50K1) *)
	WY10100_31 AT  %MX10100.31 : BOOL; (*STN 1 PROCESS TANK PUMP ON/OFF (-50K1) *)

	WY10101_00 AT  %MX10104.0 : BOOL; (*STN 2 PROCESS TANK PUMP ON/OFF (-51K1) *)
	WY10101_01 AT  %MX10104.1 : BOOL; (*STN 2 PROCESS TANK PUMP ON/OFF (-51K1) *)
	WY10101_02 AT  %MX10104.2 : BOOL; (*STN 2 PROCESS TANK PUMP ON/OFF (-51K1) *)
	WY10101_03 AT  %MX10104.3 : BOOL; (*STN 2 PROCESS TANK PUMP ON/OFF (-51K1) *)
	WY10101_04 AT  %MX10104.4 : BOOL; (*STN 2 PROCESS TANK PUMP ON/OFF (-51K1) *)
	WY10101_05 AT  %MX10104.5 : BOOL; (*STN 2 PROCESS TANK PUMP ON/OFF (-51K1) *)
	WY10101_06 AT  %MX10104.6 : BOOL; (*STN 2 PROCESS TANK PUMP ON/OFF (-51K1) *)
	WY10101_07 AT  %MX10104.7 : BOOL; (*STN 2 PROCESS TANK PUMP ON/OFF (-51K1) *)
	WY10101_08 AT  %MX10104.8 : BOOL; (*STN 2 PROCESS TANK PUMP ON/OFF (-51K1) *)
	WY10101_09 AT  %MX10104.9 : BOOL; (*STN 2 PROCESS TANK PUMP ON/OFF (-51K1) *)
	WY10101_10 AT  %MX10104.10 : BOOL; (*STN 2 PROCESS TANK PUMP ON/OFF (-51K1) *)
	WY10101_11 AT  %MX10104.11 : BOOL; (*STN 2 PROCESS TANK PUMP ON/OFF (-51K1) *)
	WY10101_12 AT  %MX10104.12 : BOOL; (*STN 2 PROCESS TANK PUMP ON/OFF (-51K1) *)
	WY10101_13 AT  %MX10104.13 : BOOL; (*STN 2 PROCESS TANK PUMP ON/OFF (-51K1) *)
	WY10101_14 AT  %MX10104.14 : BOOL; (*STN 2 PROCESS TANK PUMP ON/OFF (-51K1) *)
	WY10101_15 AT  %MX10104.15 : BOOL; (*STN 2 PROCESS TANK PUMP ON/OFF (-51K1) *)
	WY10101_16 AT  %MX10104.16 : BOOL; (*STN 2 PROCESS TANK PUMP ON/OFF (-51K1) *)
	WY10101_17 AT  %MX10104.17 : BOOL; (*STN 2 PROCESS TANK PUMP ON/OFF (-51K1) *)
	WY10101_18 AT  %MX10104.18 : BOOL; (*STN 2 PROCESS TANK PUMP ON/OFF (-51K1) *)
	WY10101_19 AT  %MX10104.19 : BOOL; (*STN 2 PROCESS TANK PUMP ON/OFF (-51K1) *)
	WY10101_20 AT  %MX10104.20 : BOOL; (*STN 2 PROCESS TANK PUMP ON/OFF (-51K1) *)
	WY10101_21 AT  %MX10104.21 : BOOL; (*STN 2 PROCESS TANK PUMP ON/OFF (-51K1) *)
	WY10101_22 AT  %MX10104.22 : BOOL; (*STN 2 PROCESS TANK PUMP ON/OFF (-51K1) *)
	WY10101_23 AT  %MX10104.23 : BOOL; (*STN 2 PROCESS TANK PUMP ON/OFF (-51K1) *)
	WY10101_24 AT  %MX10104.24 : BOOL; (*STN 2 PROCESS TANK PUMP ON/OFF (-51K1) *)
	WY10101_25 AT  %MX10104.25 : BOOL; (*STN 2 PROCESS TANK PUMP ON/OFF (-51K1) *)
	WY10101_26 AT  %MX10104.26 : BOOL; (*STN 2 PROCESS TANK PUMP ON/OFF (-51K1) *)
	WY10101_27 AT  %MX10104.27 : BOOL; (*STN 2 PROCESS TANK PUMP ON/OFF (-51K1) *)
	WY10101_28 AT  %MX10104.28 : BOOL; (*STN 2 PROCESS TANK PUMP ON/OFF (-51K1) *)
	WY10101_29 AT  %MX10104.29 : BOOL; (*STN 2 PROCESS TANK PUMP ON/OFF (-51K1) *)
	WY10101_30 AT  %MX10104.30 : BOOL; (*STN 2 PROCESS TANK PUMP ON/OFF (-51K1) *)
	WY10101_31 AT  %MX10104.31 : BOOL; (*STN 2 PROCESS TANK PUMP ON/OFF (-51K1) *)

	WY10102_00 AT  %MX10108.0 : BOOL; (*STN 3 PROCESS TANK PUMP ON/OFF (-52K1) *)
	WY10102_01 AT  %MX10108.1 : BOOL; (*STN 3 PROCESS TANK PUMP ON/OFF (-52K1) *)
	WY10102_02 AT  %MX10108.2 : BOOL; (*STN 3 PROCESS TANK PUMP ON/OFF (-52K1) *)
	WY10102_03 AT  %MX10108.3 : BOOL; (*STN 3 PROCESS TANK PUMP ON/OFF (-52K1) *)
	WY10102_04 AT  %MX10108.4 : BOOL; (*STN 3 PROCESS TANK PUMP ON/OFF (-52K1) *)
	WY10102_05 AT  %MX10108.5 : BOOL; (*STN 3 PROCESS TANK PUMP ON/OFF (-52K1) *)
	WY10102_06 AT  %MX10108.6 : BOOL; (*STN 3 PROCESS TANK PUMP ON/OFF (-52K1) *)
	WY10102_07 AT  %MX10108.7 : BOOL; (*STN 3 PROCESS TANK PUMP ON/OFF (-52K1) *)
	WY10102_08 AT  %MX10108.8 : BOOL; (*STN 3 PROCESS TANK PUMP ON/OFF (-52K1) *)
	WY10102_09 AT  %MX10108.9 : BOOL; (*STN 3 PROCESS TANK PUMP ON/OFF (-52K1) *)
	WY10102_10 AT  %MX10108.10 : BOOL; (*STN 3 PROCESS TANK PUMP ON/OFF (-52K1) *)
	WY10102_11 AT  %MX10108.11 : BOOL; (*STN 3 PROCESS TANK PUMP ON/OFF (-52K1) *)
	WY10102_12 AT  %MX10108.12 : BOOL; (*STN 3 PROCESS TANK PUMP ON/OFF (-52K1) *)
	WY10102_13 AT  %MX10108.13 : BOOL; (*STN 3 PROCESS TANK PUMP ON/OFF (-52K1) *)
	WY10102_14 AT  %MX10108.14 : BOOL; (*STN 3 PROCESS TANK PUMP ON/OFF (-52K1) *)
	WY10102_15 AT  %MX10108.15 : BOOL; (*STN 3 PROCESS TANK PUMP ON/OFF (-52K1) *)
	WY10102_16 AT  %MX10108.16 : BOOL; (*STN 3 PROCESS TANK PUMP ON/OFF (-52K1) *)
	WY10102_17 AT  %MX10108.17 : BOOL; (*STN 3 PROCESS TANK PUMP ON/OFF (-52K1) *)
	WY10102_18 AT  %MX10108.18 : BOOL; (*STN 3 PROCESS TANK PUMP ON/OFF (-52K1) *)
	WY10102_19 AT  %MX10108.19 : BOOL; (*STN 3 PROCESS TANK PUMP ON/OFF (-52K1) *)
	WY10102_20 AT  %MX10108.20 : BOOL; (*STN 3 PROCESS TANK PUMP ON/OFF (-52K1) *)
	WY10102_21 AT  %MX10108.21 : BOOL; (*STN 3 PROCESS TANK PUMP ON/OFF (-52K1) *)
	WY10102_22 AT  %MX10108.22 : BOOL; (*STN 3 PROCESS TANK PUMP ON/OFF (-52K1) *)
	WY10102_23 AT  %MX10108.23 : BOOL; (*STN 3 PROCESS TANK PUMP ON/OFF (-52K1) *)
	WY10102_24 AT  %MX10108.24 : BOOL; (*STN 3 PROCESS TANK PUMP ON/OFF (-52K1) *)
	WY10102_25 AT  %MX10108.25 : BOOL; (*STN 3 PROCESS TANK PUMP ON/OFF (-52K1) *)
	WY10102_26 AT  %MX10108.26 : BOOL; (*STN 3 PROCESS TANK PUMP ON/OFF (-52K1) *)
	WY10102_27 AT  %MX10108.27 : BOOL; (*STN 3 PROCESS TANK PUMP ON/OFF (-52K1) *)
	WY10102_28 AT  %MX10108.28 : BOOL; (*STN 3 PROCESS TANK PUMP ON/OFF (-52K1) *)
	WY10102_29 AT  %MX10108.29 : BOOL; (*STN 3 PROCESS TANK PUMP ON/OFF (-52K1) *)
	WY10102_30 AT  %MX10108.30 : BOOL; (*STN 3 PROCESS TANK PUMP ON/OFF (-52K1) *)
	WY10102_31 AT  %MX10108.31 : BOOL; (*STN 3 PROCESS TANK PUMP ON/OFF (-52K1) *)

	WY10103_00 AT  %MX10112.0 : BOOL; (*STN 5 VACUUM PUMP ON/OFF (-56K1) *)
	WY10103_01 AT  %MX10112.1 : BOOL; (*STN 5 VACUUM PUMP ON/OFF (-56K1) *)
	WY10103_02 AT  %MX10112.2 : BOOL; (*STN 5 VACUUM PUMP ON/OFF (-56K1) *)
	WY10103_03 AT  %MX10112.3 : BOOL; (*STN 5 VACUUM PUMP ON/OFF (-56K1) *)
	WY10103_04 AT  %MX10112.4 : BOOL; (*STN 5 VACUUM PUMP ON/OFF (-56K1) *)
	WY10103_05 AT  %MX10112.5 : BOOL; (*STN 5 VACUUM PUMP ON/OFF (-56K1) *)
	WY10103_06 AT  %MX10112.6 : BOOL; (*STN 5 VACUUM PUMP ON/OFF (-56K1) *)
	WY10103_07 AT  %MX10112.7 : BOOL; (*STN 5 VACUUM PUMP ON/OFF (-56K1) *)
	WY10103_08 AT  %MX10112.8 : BOOL; (*STN 5 VACUUM PUMP ON/OFF (-56K1) *)
	WY10103_09 AT  %MX10112.9 : BOOL; (*STN 5 VACUUM PUMP ON/OFF (-56K1) *)
	WY10103_10 AT  %MX10112.10 : BOOL; (*STN 5 VACUUM PUMP ON/OFF (-56K1) *)
	WY10103_11 AT  %MX10112.11 : BOOL; (*STN 5 VACUUM PUMP ON/OFF (-56K1) *)
	WY10103_12 AT  %MX10112.12 : BOOL; (*STN 5 VACUUM PUMP ON/OFF (-56K1) *)
	WY10103_13 AT  %MX10112.13 : BOOL; (*STN 5 VACUUM PUMP ON/OFF (-56K1) *)
	WY10103_14 AT  %MX10112.14 : BOOL; (*STN 5 VACUUM PUMP ON/OFF (-56K1) *)
	WY10103_15 AT  %MX10112.15 : BOOL; (*STN 5 VACUUM PUMP ON/OFF (-56K1) *)
	WY10103_16 AT  %MX10112.16 : BOOL; (*STN 5 VACUUM PUMP ON/OFF (-56K1) *)
	WY10103_17 AT  %MX10112.17 : BOOL; (*STN 5 VACUUM PUMP ON/OFF (-56K1) *)
	WY10103_18 AT  %MX10112.18 : BOOL; (*STN 5 VACUUM PUMP ON/OFF (-56K1) *)
	WY10103_19 AT  %MX10112.19 : BOOL; (*STN 5 VACUUM PUMP ON/OFF (-56K1) *)
	WY10103_20 AT  %MX10112.20 : BOOL; (*STN 5 VACUUM PUMP ON/OFF (-56K1) *)
	WY10103_21 AT  %MX10112.21 : BOOL; (*STN 5 VACUUM PUMP ON/OFF (-56K1) *)
	WY10103_22 AT  %MX10112.22 : BOOL; (*STN 5 VACUUM PUMP ON/OFF (-56K1) *)
	WY10103_23 AT  %MX10112.23 : BOOL; (*STN 5 VACUUM PUMP ON/OFF (-56K1) *)
	WY10103_24 AT  %MX10112.24 : BOOL; (*STN 5 VACUUM PUMP ON/OFF (-56K1) *)
	WY10103_25 AT  %MX10112.25 : BOOL; (*STN 5 VACUUM PUMP ON/OFF (-56K1) *)
	WY10103_26 AT  %MX10112.26 : BOOL; (*STN 5 VACUUM PUMP ON/OFF (-56K1) *)
	WY10103_27 AT  %MX10112.27 : BOOL; (*STN 5 VACUUM PUMP ON/OFF (-56K1) *)
	WY10103_28 AT  %MX10112.28 : BOOL; (*STN 5 VACUUM PUMP ON/OFF (-56K1) *)
	WY10103_29 AT  %MX10112.29 : BOOL; (*STN 5 VACUUM PUMP ON/OFF (-56K1) *)
	WY10103_30 AT  %MX10112.30 : BOOL; (*STN 5 VACUUM PUMP ON/OFF (-56K1) *)
	WY10103_31 AT  %MX10112.31 : BOOL; (*STN 5 VACUUM PUMP ON/OFF (-56K1) *)

	WY10104_00 AT  %MX10116.0 : BOOL; (*STN 2&3 AGITATION MOTOR ON/OFF (-25K1) *)
	WY10104_01 AT  %MX10116.1 : BOOL; (*STN 2&3 AGITATION MOTOR ON/OFF (-25K1) *)
	WY10104_02 AT  %MX10116.2 : BOOL; (*STN 2&3 AGITATION MOTOR ON/OFF (-25K1) *)
	WY10104_03 AT  %MX10116.3 : BOOL; (*STN 2&3 AGITATION MOTOR ON/OFF (-25K1) *)
	WY10104_04 AT  %MX10116.4 : BOOL; (*STN 2&3 AGITATION MOTOR ON/OFF (-25K1) *)
	WY10104_05 AT  %MX10116.5 : BOOL; (*STN 2&3 AGITATION MOTOR ON/OFF (-25K1) *)
	WY10104_06 AT  %MX10116.6 : BOOL; (*STN 2&3 AGITATION MOTOR ON/OFF (-25K1) *)
	WY10104_07 AT  %MX10116.7 : BOOL; (*STN 2&3 AGITATION MOTOR ON/OFF (-25K1) *)
	WY10104_08 AT  %MX10116.8 : BOOL; (*STN 2&3 AGITATION MOTOR ON/OFF (-25K1) *)
	WY10104_09 AT  %MX10116.9 : BOOL; (*STN 2&3 AGITATION MOTOR ON/OFF (-25K1) *)
	WY10104_10 AT  %MX10116.10 : BOOL; (*STN 2&3 AGITATION MOTOR ON/OFF (-25K1) *)
	WY10104_11 AT  %MX10116.11 : BOOL; (*STN 2&3 AGITATION MOTOR ON/OFF (-25K1) *)
	WY10104_12 AT  %MX10116.12 : BOOL; (*STN 2&3 AGITATION MOTOR ON/OFF (-25K1) *)
	WY10104_13 AT  %MX10116.13 : BOOL; (*STN 2&3 AGITATION MOTOR ON/OFF (-25K1) *)
	WY10104_14 AT  %MX10116.14 : BOOL; (*STN 2&3 AGITATION MOTOR ON/OFF (-25K1) *)
	WY10104_15 AT  %MX10116.15 : BOOL; (*STN 2&3 AGITATION MOTOR ON/OFF (-25K1) *)
	WY10104_16 AT  %MX10116.16 : BOOL; (*STN 2&3 AGITATION MOTOR ON/OFF (-25K1) *)
	WY10104_17 AT  %MX10116.17 : BOOL; (*STN 2&3 AGITATION MOTOR ON/OFF (-25K1) *)
	WY10104_18 AT  %MX10116.18 : BOOL; (*STN 2&3 AGITATION MOTOR ON/OFF (-25K1) *)
	WY10104_19 AT  %MX10116.19 : BOOL; (*STN 2&3 AGITATION MOTOR ON/OFF (-25K1) *)
	WY10104_20 AT  %MX10116.20 : BOOL; (*STN 2&3 AGITATION MOTOR ON/OFF (-25K1) *)
	WY10104_21 AT  %MX10116.21 : BOOL; (*STN 2&3 AGITATION MOTOR ON/OFF (-25K1) *)
	WY10104_22 AT  %MX10116.22 : BOOL; (*STN 2&3 AGITATION MOTOR ON/OFF (-25K1) *)
	WY10104_23 AT  %MX10116.23 : BOOL; (*STN 2&3 AGITATION MOTOR ON/OFF (-25K1) *)
	WY10104_24 AT  %MX10116.24 : BOOL; (*STN 2&3 AGITATION MOTOR ON/OFF (-25K1) *)
	WY10104_25 AT  %MX10116.25 : BOOL; (*STN 2&3 AGITATION MOTOR ON/OFF (-25K1) *)
	WY10104_26 AT  %MX10116.26 : BOOL; (*STN 2&3 AGITATION MOTOR ON/OFF (-25K1) *)
	WY10104_27 AT  %MX10116.27 : BOOL; (*STN 2&3 AGITATION MOTOR ON/OFF (-25K1) *)
	WY10104_28 AT  %MX10116.28 : BOOL; (*STN 2&3 AGITATION MOTOR ON/OFF (-25K1) *)
	WY10104_29 AT  %MX10116.29 : BOOL; (*STN 2&3 AGITATION MOTOR ON/OFF (-25K1) *)
	WY10104_30 AT  %MX10116.30 : BOOL; (*STN 2&3 AGITATION MOTOR ON/OFF (-25K1) *)
	WY10104_31 AT  %MX10116.31 : BOOL; (*STN 2&3 AGITATION MOTOR ON/OFF (-25K1) *)

	WY10105_00 AT  %MX10120.0 : BOOL; (*STN 5 BLOWER ON/OFF (-65K1) *)
	WY10105_01 AT  %MX10120.1 : BOOL; (*STN 5 BLOWER ON/OFF (-65K1) *)
	WY10105_02 AT  %MX10120.2 : BOOL; (*STN 5 BLOWER ON/OFF (-65K1) *)
	WY10105_03 AT  %MX10120.3 : BOOL; (*STN 5 BLOWER ON/OFF (-65K1) *)
	WY10105_04 AT  %MX10120.4 : BOOL; (*STN 5 BLOWER ON/OFF (-65K1) *)
	WY10105_05 AT  %MX10120.5 : BOOL; (*STN 5 BLOWER ON/OFF (-65K1) *)
	WY10105_06 AT  %MX10120.6 : BOOL; (*STN 5 BLOWER ON/OFF (-65K1) *)
	WY10105_07 AT  %MX10120.7 : BOOL; (*STN 5 BLOWER ON/OFF (-65K1) *)
	WY10105_08 AT  %MX10120.8 : BOOL; (*STN 5 BLOWER ON/OFF (-65K1) *)
	WY10105_09 AT  %MX10120.9 : BOOL; (*STN 5 BLOWER ON/OFF (-65K1) *)
	WY10105_10 AT  %MX10120.10 : BOOL; (*STN 5 BLOWER ON/OFF (-65K1) *)
	WY10105_11 AT  %MX10120.11 : BOOL; (*STN 5 BLOWER ON/OFF (-65K1) *)
	WY10105_12 AT  %MX10120.12 : BOOL; (*STN 5 BLOWER ON/OFF (-65K1) *)
	WY10105_13 AT  %MX10120.13 : BOOL; (*STN 5 BLOWER ON/OFF (-65K1) *)
	WY10105_14 AT  %MX10120.14 : BOOL; (*STN 5 BLOWER ON/OFF (-65K1) *)
	WY10105_15 AT  %MX10120.15 : BOOL; (*STN 5 BLOWER ON/OFF (-65K1) *)
	WY10105_16 AT  %MX10120.16 : BOOL; (*STN 5 BLOWER ON/OFF (-65K1) *)
	WY10105_17 AT  %MX10120.17 : BOOL; (*STN 5 BLOWER ON/OFF (-65K1) *)
	WY10105_18 AT  %MX10120.18 : BOOL; (*STN 5 BLOWER ON/OFF (-65K1) *)
	WY10105_19 AT  %MX10120.19 : BOOL; (*STN 5 BLOWER ON/OFF (-65K1) *)
	WY10105_20 AT  %MX10120.20 : BOOL; (*STN 5 BLOWER ON/OFF (-65K1) *)
	WY10105_21 AT  %MX10120.21 : BOOL; (*STN 5 BLOWER ON/OFF (-65K1) *)
	WY10105_22 AT  %MX10120.22 : BOOL; (*STN 5 BLOWER ON/OFF (-65K1) *)
	WY10105_23 AT  %MX10120.23 : BOOL; (*STN 5 BLOWER ON/OFF (-65K1) *)
	WY10105_24 AT  %MX10120.24 : BOOL; (*STN 5 BLOWER ON/OFF (-65K1) *)
	WY10105_25 AT  %MX10120.25 : BOOL; (*STN 5 BLOWER ON/OFF (-65K1) *)
	WY10105_26 AT  %MX10120.26 : BOOL; (*STN 5 BLOWER ON/OFF (-65K1) *)
	WY10105_27 AT  %MX10120.27 : BOOL; (*STN 5 BLOWER ON/OFF (-65K1) *)
	WY10105_28 AT  %MX10120.28 : BOOL; (*STN 5 BLOWER ON/OFF (-65K1) *)
	WY10105_29 AT  %MX10120.29 : BOOL; (*STN 5 BLOWER ON/OFF (-65K1) *)
	WY10105_30 AT  %MX10120.30 : BOOL; (*STN 5 BLOWER ON/OFF (-65K1) *)
	WY10105_31 AT  %MX10120.31 : BOOL; (*STN 5 BLOWER ON/OFF (-65K1) *)

	WY10106_00 AT  %MX10124.0 : BOOL; (*STN 1 SUB PROCESS TANK STIRRING MOTOR ON/OFF (-26K1) *)
	WY10106_01 AT  %MX10124.1 : BOOL; (*STN 1 SUB PROCESS TANK STIRRING MOTOR ON/OFF (-26K1) *)
	WY10106_02 AT  %MX10124.2 : BOOL; (*STN 1 SUB PROCESS TANK STIRRING MOTOR ON/OFF (-26K1) *)
	WY10106_03 AT  %MX10124.3 : BOOL; (*STN 1 SUB PROCESS TANK STIRRING MOTOR ON/OFF (-26K1) *)
	WY10106_04 AT  %MX10124.4 : BOOL; (*STN 1 SUB PROCESS TANK STIRRING MOTOR ON/OFF (-26K1) *)
	WY10106_05 AT  %MX10124.5 : BOOL; (*STN 1 SUB PROCESS TANK STIRRING MOTOR ON/OFF (-26K1) *)
	WY10106_06 AT  %MX10124.6 : BOOL; (*STN 1 SUB PROCESS TANK STIRRING MOTOR ON/OFF (-26K1) *)
	WY10106_07 AT  %MX10124.7 : BOOL; (*STN 1 SUB PROCESS TANK STIRRING MOTOR ON/OFF (-26K1) *)
	WY10106_08 AT  %MX10124.8 : BOOL; (*STN 1 SUB PROCESS TANK STIRRING MOTOR ON/OFF (-26K1) *)
	WY10106_09 AT  %MX10124.9 : BOOL; (*STN 1 SUB PROCESS TANK STIRRING MOTOR ON/OFF (-26K1) *)
	WY10106_10 AT  %MX10124.10 : BOOL; (*STN 1 SUB PROCESS TANK STIRRING MOTOR ON/OFF (-26K1) *)
	WY10106_11 AT  %MX10124.11 : BOOL; (*STN 1 SUB PROCESS TANK STIRRING MOTOR ON/OFF (-26K1) *)
	WY10106_12 AT  %MX10124.12 : BOOL; (*STN 1 SUB PROCESS TANK STIRRING MOTOR ON/OFF (-26K1) *)
	WY10106_13 AT  %MX10124.13 : BOOL; (*STN 1 SUB PROCESS TANK STIRRING MOTOR ON/OFF (-26K1) *)
	WY10106_14 AT  %MX10124.14 : BOOL; (*STN 1 SUB PROCESS TANK STIRRING MOTOR ON/OFF (-26K1) *)
	WY10106_15 AT  %MX10124.15 : BOOL; (*STN 1 SUB PROCESS TANK STIRRING MOTOR ON/OFF (-26K1) *)
	WY10106_16 AT  %MX10124.16 : BOOL; (*STN 1 SUB PROCESS TANK STIRRING MOTOR ON/OFF (-26K1) *)
	WY10106_17 AT  %MX10124.17 : BOOL; (*STN 1 SUB PROCESS TANK STIRRING MOTOR ON/OFF (-26K1) *)
	WY10106_18 AT  %MX10124.18 : BOOL; (*STN 1 SUB PROCESS TANK STIRRING MOTOR ON/OFF (-26K1) *)
	WY10106_19 AT  %MX10124.19 : BOOL; (*STN 1 SUB PROCESS TANK STIRRING MOTOR ON/OFF (-26K1) *)
	WY10106_20 AT  %MX10124.20 : BOOL; (*STN 1 SUB PROCESS TANK STIRRING MOTOR ON/OFF (-26K1) *)
	WY10106_21 AT  %MX10124.21 : BOOL; (*STN 1 SUB PROCESS TANK STIRRING MOTOR ON/OFF (-26K1) *)
	WY10106_22 AT  %MX10124.22 : BOOL; (*STN 1 SUB PROCESS TANK STIRRING MOTOR ON/OFF (-26K1) *)
	WY10106_23 AT  %MX10124.23 : BOOL; (*STN 1 SUB PROCESS TANK STIRRING MOTOR ON/OFF (-26K1) *)
	WY10106_24 AT  %MX10124.24 : BOOL; (*STN 1 SUB PROCESS TANK STIRRING MOTOR ON/OFF (-26K1) *)
	WY10106_25 AT  %MX10124.25 : BOOL; (*STN 1 SUB PROCESS TANK STIRRING MOTOR ON/OFF (-26K1) *)
	WY10106_26 AT  %MX10124.26 : BOOL; (*STN 1 SUB PROCESS TANK STIRRING MOTOR ON/OFF (-26K1) *)
	WY10106_27 AT  %MX10124.27 : BOOL; (*STN 1 SUB PROCESS TANK STIRRING MOTOR ON/OFF (-26K1) *)
	WY10106_28 AT  %MX10124.28 : BOOL; (*STN 1 SUB PROCESS TANK STIRRING MOTOR ON/OFF (-26K1) *)
	WY10106_29 AT  %MX10124.29 : BOOL; (*STN 1 SUB PROCESS TANK STIRRING MOTOR ON/OFF (-26K1) *)
	WY10106_30 AT  %MX10124.30 : BOOL; (*STN 1 SUB PROCESS TANK STIRRING MOTOR ON/OFF (-26K1) *)
	WY10106_31 AT  %MX10124.31 : BOOL; (*STN 1 SUB PROCESS TANK STIRRING MOTOR ON/OFF (-26K1) *)

	WY10107_00 AT  %MX10128.0 : BOOL; (*DETERGENT TANK 1 STIRRING MOTOR ON/OFF (-27K1) *)
	WY10107_01 AT  %MX10128.1 : BOOL; (*DETERGENT TANK 1 STIRRING MOTOR ON/OFF (-27K1) *)
	WY10107_02 AT  %MX10128.2 : BOOL; (*DETERGENT TANK 1 STIRRING MOTOR ON/OFF (-27K1) *)
	WY10107_03 AT  %MX10128.3 : BOOL; (*DETERGENT TANK 1 STIRRING MOTOR ON/OFF (-27K1) *)
	WY10107_04 AT  %MX10128.4 : BOOL; (*DETERGENT TANK 1 STIRRING MOTOR ON/OFF (-27K1) *)
	WY10107_05 AT  %MX10128.5 : BOOL; (*DETERGENT TANK 1 STIRRING MOTOR ON/OFF (-27K1) *)
	WY10107_06 AT  %MX10128.6 : BOOL; (*DETERGENT TANK 1 STIRRING MOTOR ON/OFF (-27K1) *)
	WY10107_07 AT  %MX10128.7 : BOOL; (*DETERGENT TANK 1 STIRRING MOTOR ON/OFF (-27K1) *)
	WY10107_08 AT  %MX10128.8 : BOOL; (*DETERGENT TANK 1 STIRRING MOTOR ON/OFF (-27K1) *)
	WY10107_09 AT  %MX10128.9 : BOOL; (*DETERGENT TANK 1 STIRRING MOTOR ON/OFF (-27K1) *)
	WY10107_10 AT  %MX10128.10 : BOOL; (*DETERGENT TANK 1 STIRRING MOTOR ON/OFF (-27K1) *)
	WY10107_11 AT  %MX10128.11 : BOOL; (*DETERGENT TANK 1 STIRRING MOTOR ON/OFF (-27K1) *)
	WY10107_12 AT  %MX10128.12 : BOOL; (*DETERGENT TANK 1 STIRRING MOTOR ON/OFF (-27K1) *)
	WY10107_13 AT  %MX10128.13 : BOOL; (*DETERGENT TANK 1 STIRRING MOTOR ON/OFF (-27K1) *)
	WY10107_14 AT  %MX10128.14 : BOOL; (*DETERGENT TANK 1 STIRRING MOTOR ON/OFF (-27K1) *)
	WY10107_15 AT  %MX10128.15 : BOOL; (*DETERGENT TANK 1 STIRRING MOTOR ON/OFF (-27K1) *)
	WY10107_16 AT  %MX10128.16 : BOOL; (*DETERGENT TANK 1 STIRRING MOTOR ON/OFF (-27K1) *)
	WY10107_17 AT  %MX10128.17 : BOOL; (*DETERGENT TANK 1 STIRRING MOTOR ON/OFF (-27K1) *)
	WY10107_18 AT  %MX10128.18 : BOOL; (*DETERGENT TANK 1 STIRRING MOTOR ON/OFF (-27K1) *)
	WY10107_19 AT  %MX10128.19 : BOOL; (*DETERGENT TANK 1 STIRRING MOTOR ON/OFF (-27K1) *)
	WY10107_20 AT  %MX10128.20 : BOOL; (*DETERGENT TANK 1 STIRRING MOTOR ON/OFF (-27K1) *)
	WY10107_21 AT  %MX10128.21 : BOOL; (*DETERGENT TANK 1 STIRRING MOTOR ON/OFF (-27K1) *)
	WY10107_22 AT  %MX10128.22 : BOOL; (*DETERGENT TANK 1 STIRRING MOTOR ON/OFF (-27K1) *)
	WY10107_23 AT  %MX10128.23 : BOOL; (*DETERGENT TANK 1 STIRRING MOTOR ON/OFF (-27K1) *)
	WY10107_24 AT  %MX10128.24 : BOOL; (*DETERGENT TANK 1 STIRRING MOTOR ON/OFF (-27K1) *)
	WY10107_25 AT  %MX10128.25 : BOOL; (*DETERGENT TANK 1 STIRRING MOTOR ON/OFF (-27K1) *)
	WY10107_26 AT  %MX10128.26 : BOOL; (*DETERGENT TANK 1 STIRRING MOTOR ON/OFF (-27K1) *)
	WY10107_27 AT  %MX10128.27 : BOOL; (*DETERGENT TANK 1 STIRRING MOTOR ON/OFF (-27K1) *)
	WY10107_28 AT  %MX10128.28 : BOOL; (*DETERGENT TANK 1 STIRRING MOTOR ON/OFF (-27K1) *)
	WY10107_29 AT  %MX10128.29 : BOOL; (*DETERGENT TANK 1 STIRRING MOTOR ON/OFF (-27K1) *)
	WY10107_30 AT  %MX10128.30 : BOOL; (*DETERGENT TANK 1 STIRRING MOTOR ON/OFF (-27K1) *)
	WY10107_31 AT  %MX10128.31 : BOOL; (*DETERGENT TANK 1 STIRRING MOTOR ON/OFF (-27K1) *)

	WY10108_00 AT  %MX10132.0 : BOOL; (*STN 1 ULTRASONIC ON/OFF (-16K1) *)
	WY10108_01 AT  %MX10132.1 : BOOL; (*STN 1 ULTRASONIC ON/OFF (-16K1) *)
	WY10108_02 AT  %MX10132.2 : BOOL; (*STN 1 ULTRASONIC ON/OFF (-16K1) *)
	WY10108_03 AT  %MX10132.3 : BOOL; (*STN 1 ULTRASONIC ON/OFF (-16K1) *)
	WY10108_04 AT  %MX10132.4 : BOOL; (*STN 1 ULTRASONIC ON/OFF (-16K1) *)
	WY10108_05 AT  %MX10132.5 : BOOL; (*STN 1 ULTRASONIC ON/OFF (-16K1) *)
	WY10108_06 AT  %MX10132.6 : BOOL; (*STN 1 ULTRASONIC ON/OFF (-16K1) *)
	WY10108_07 AT  %MX10132.7 : BOOL; (*STN 1 ULTRASONIC ON/OFF (-16K1) *)
	WY10108_08 AT  %MX10132.8 : BOOL; (*STN 1 ULTRASONIC ON/OFF (-16K1) *)
	WY10108_09 AT  %MX10132.9 : BOOL; (*STN 1 ULTRASONIC ON/OFF (-16K1) *)
	WY10108_10 AT  %MX10132.10 : BOOL; (*STN 1 ULTRASONIC ON/OFF (-16K1) *)
	WY10108_11 AT  %MX10132.11 : BOOL; (*STN 1 ULTRASONIC ON/OFF (-16K1) *)
	WY10108_12 AT  %MX10132.12 : BOOL; (*STN 1 ULTRASONIC ON/OFF (-16K1) *)
	WY10108_13 AT  %MX10132.13 : BOOL; (*STN 1 ULTRASONIC ON/OFF (-16K1) *)
	WY10108_14 AT  %MX10132.14 : BOOL; (*STN 1 ULTRASONIC ON/OFF (-16K1) *)
	WY10108_15 AT  %MX10132.15 : BOOL; (*STN 1 ULTRASONIC ON/OFF (-16K1) *)
	WY10108_16 AT  %MX10132.16 : BOOL; (*STN 1 ULTRASONIC ON/OFF (-16K1) *)
	WY10108_17 AT  %MX10132.17 : BOOL; (*STN 1 ULTRASONIC ON/OFF (-16K1) *)
	WY10108_18 AT  %MX10132.18 : BOOL; (*STN 1 ULTRASONIC ON/OFF (-16K1) *)
	WY10108_19 AT  %MX10132.19 : BOOL; (*STN 1 ULTRASONIC ON/OFF (-16K1) *)
	WY10108_20 AT  %MX10132.20 : BOOL; (*STN 1 ULTRASONIC ON/OFF (-16K1) *)
	WY10108_21 AT  %MX10132.21 : BOOL; (*STN 1 ULTRASONIC ON/OFF (-16K1) *)
	WY10108_22 AT  %MX10132.22 : BOOL; (*STN 1 ULTRASONIC ON/OFF (-16K1) *)
	WY10108_23 AT  %MX10132.23 : BOOL; (*STN 1 ULTRASONIC ON/OFF (-16K1) *)
	WY10108_24 AT  %MX10132.24 : BOOL; (*STN 1 ULTRASONIC ON/OFF (-16K1) *)
	WY10108_25 AT  %MX10132.25 : BOOL; (*STN 1 ULTRASONIC ON/OFF (-16K1) *)
	WY10108_26 AT  %MX10132.26 : BOOL; (*STN 1 ULTRASONIC ON/OFF (-16K1) *)
	WY10108_27 AT  %MX10132.27 : BOOL; (*STN 1 ULTRASONIC ON/OFF (-16K1) *)
	WY10108_28 AT  %MX10132.28 : BOOL; (*STN 1 ULTRASONIC ON/OFF (-16K1) *)
	WY10108_29 AT  %MX10132.29 : BOOL; (*STN 1 ULTRASONIC ON/OFF (-16K1) *)
	WY10108_30 AT  %MX10132.30 : BOOL; (*STN 1 ULTRASONIC ON/OFF (-16K1) *)
	WY10108_31 AT  %MX10132.31 : BOOL; (*STN 1 ULTRASONIC ON/OFF (-16K1) *)

	WY10109_00 AT  %MX10136.0 : BOOL; (*STN 2 ULTRASONIC ON/OFF (-17K1) *)
	WY10109_01 AT  %MX10136.1 : BOOL; (*STN 2 ULTRASONIC ON/OFF (-17K1) *)
	WY10109_02 AT  %MX10136.2 : BOOL; (*STN 2 ULTRASONIC ON/OFF (-17K1) *)
	WY10109_03 AT  %MX10136.3 : BOOL; (*STN 2 ULTRASONIC ON/OFF (-17K1) *)
	WY10109_04 AT  %MX10136.4 : BOOL; (*STN 2 ULTRASONIC ON/OFF (-17K1) *)
	WY10109_05 AT  %MX10136.5 : BOOL; (*STN 2 ULTRASONIC ON/OFF (-17K1) *)
	WY10109_06 AT  %MX10136.6 : BOOL; (*STN 2 ULTRASONIC ON/OFF (-17K1) *)
	WY10109_07 AT  %MX10136.7 : BOOL; (*STN 2 ULTRASONIC ON/OFF (-17K1) *)
	WY10109_08 AT  %MX10136.8 : BOOL; (*STN 2 ULTRASONIC ON/OFF (-17K1) *)
	WY10109_09 AT  %MX10136.9 : BOOL; (*STN 2 ULTRASONIC ON/OFF (-17K1) *)
	WY10109_10 AT  %MX10136.10 : BOOL; (*STN 2 ULTRASONIC ON/OFF (-17K1) *)
	WY10109_11 AT  %MX10136.11 : BOOL; (*STN 2 ULTRASONIC ON/OFF (-17K1) *)
	WY10109_12 AT  %MX10136.12 : BOOL; (*STN 2 ULTRASONIC ON/OFF (-17K1) *)
	WY10109_13 AT  %MX10136.13 : BOOL; (*STN 2 ULTRASONIC ON/OFF (-17K1) *)
	WY10109_14 AT  %MX10136.14 : BOOL; (*STN 2 ULTRASONIC ON/OFF (-17K1) *)
	WY10109_15 AT  %MX10136.15 : BOOL; (*STN 2 ULTRASONIC ON/OFF (-17K1) *)
	WY10109_16 AT  %MX10136.16 : BOOL; (*STN 2 ULTRASONIC ON/OFF (-17K1) *)
	WY10109_17 AT  %MX10136.17 : BOOL; (*STN 2 ULTRASONIC ON/OFF (-17K1) *)
	WY10109_18 AT  %MX10136.18 : BOOL; (*STN 2 ULTRASONIC ON/OFF (-17K1) *)
	WY10109_19 AT  %MX10136.19 : BOOL; (*STN 2 ULTRASONIC ON/OFF (-17K1) *)
	WY10109_20 AT  %MX10136.20 : BOOL; (*STN 2 ULTRASONIC ON/OFF (-17K1) *)
	WY10109_21 AT  %MX10136.21 : BOOL; (*STN 2 ULTRASONIC ON/OFF (-17K1) *)
	WY10109_22 AT  %MX10136.22 : BOOL; (*STN 2 ULTRASONIC ON/OFF (-17K1) *)
	WY10109_23 AT  %MX10136.23 : BOOL; (*STN 2 ULTRASONIC ON/OFF (-17K1) *)
	WY10109_24 AT  %MX10136.24 : BOOL; (*STN 2 ULTRASONIC ON/OFF (-17K1) *)
	WY10109_25 AT  %MX10136.25 : BOOL; (*STN 2 ULTRASONIC ON/OFF (-17K1) *)
	WY10109_26 AT  %MX10136.26 : BOOL; (*STN 2 ULTRASONIC ON/OFF (-17K1) *)
	WY10109_27 AT  %MX10136.27 : BOOL; (*STN 2 ULTRASONIC ON/OFF (-17K1) *)
	WY10109_28 AT  %MX10136.28 : BOOL; (*STN 2 ULTRASONIC ON/OFF (-17K1) *)
	WY10109_29 AT  %MX10136.29 : BOOL; (*STN 2 ULTRASONIC ON/OFF (-17K1) *)
	WY10109_30 AT  %MX10136.30 : BOOL; (*STN 2 ULTRASONIC ON/OFF (-17K1) *)
	WY10109_31 AT  %MX10136.31 : BOOL; (*STN 2 ULTRASONIC ON/OFF (-17K1) *)

	WY10110_00 AT  %MX10140.0 : BOOL; (*STN 3 ULTRASONIC ON/OFF (-18K1) *)
	WY10110_01 AT  %MX10140.1 : BOOL; (*STN 3 ULTRASONIC ON/OFF (-18K1) *)
	WY10110_02 AT  %MX10140.2 : BOOL; (*STN 3 ULTRASONIC ON/OFF (-18K1) *)
	WY10110_03 AT  %MX10140.3 : BOOL; (*STN 3 ULTRASONIC ON/OFF (-18K1) *)
	WY10110_04 AT  %MX10140.4 : BOOL; (*STN 3 ULTRASONIC ON/OFF (-18K1) *)
	WY10110_05 AT  %MX10140.5 : BOOL; (*STN 3 ULTRASONIC ON/OFF (-18K1) *)
	WY10110_06 AT  %MX10140.6 : BOOL; (*STN 3 ULTRASONIC ON/OFF (-18K1) *)
	WY10110_07 AT  %MX10140.7 : BOOL; (*STN 3 ULTRASONIC ON/OFF (-18K1) *)
	WY10110_08 AT  %MX10140.8 : BOOL; (*STN 3 ULTRASONIC ON/OFF (-18K1) *)
	WY10110_09 AT  %MX10140.9 : BOOL; (*STN 3 ULTRASONIC ON/OFF (-18K1) *)
	WY10110_10 AT  %MX10140.10 : BOOL; (*STN 3 ULTRASONIC ON/OFF (-18K1) *)
	WY10110_11 AT  %MX10140.11 : BOOL; (*STN 3 ULTRASONIC ON/OFF (-18K1) *)
	WY10110_12 AT  %MX10140.12 : BOOL; (*STN 3 ULTRASONIC ON/OFF (-18K1) *)
	WY10110_13 AT  %MX10140.13 : BOOL; (*STN 3 ULTRASONIC ON/OFF (-18K1) *)
	WY10110_14 AT  %MX10140.14 : BOOL; (*STN 3 ULTRASONIC ON/OFF (-18K1) *)
	WY10110_15 AT  %MX10140.15 : BOOL; (*STN 3 ULTRASONIC ON/OFF (-18K1) *)
	WY10110_16 AT  %MX10140.16 : BOOL; (*STN 3 ULTRASONIC ON/OFF (-18K1) *)
	WY10110_17 AT  %MX10140.17 : BOOL; (*STN 3 ULTRASONIC ON/OFF (-18K1) *)
	WY10110_18 AT  %MX10140.18 : BOOL; (*STN 3 ULTRASONIC ON/OFF (-18K1) *)
	WY10110_19 AT  %MX10140.19 : BOOL; (*STN 3 ULTRASONIC ON/OFF (-18K1) *)
	WY10110_20 AT  %MX10140.20 : BOOL; (*STN 3 ULTRASONIC ON/OFF (-18K1) *)
	WY10110_21 AT  %MX10140.21 : BOOL; (*STN 3 ULTRASONIC ON/OFF (-18K1) *)
	WY10110_22 AT  %MX10140.22 : BOOL; (*STN 3 ULTRASONIC ON/OFF (-18K1) *)
	WY10110_23 AT  %MX10140.23 : BOOL; (*STN 3 ULTRASONIC ON/OFF (-18K1) *)
	WY10110_24 AT  %MX10140.24 : BOOL; (*STN 3 ULTRASONIC ON/OFF (-18K1) *)
	WY10110_25 AT  %MX10140.25 : BOOL; (*STN 3 ULTRASONIC ON/OFF (-18K1) *)
	WY10110_26 AT  %MX10140.26 : BOOL; (*STN 3 ULTRASONIC ON/OFF (-18K1) *)
	WY10110_27 AT  %MX10140.27 : BOOL; (*STN 3 ULTRASONIC ON/OFF (-18K1) *)
	WY10110_28 AT  %MX10140.28 : BOOL; (*STN 3 ULTRASONIC ON/OFF (-18K1) *)
	WY10110_29 AT  %MX10140.29 : BOOL; (*STN 3 ULTRASONIC ON/OFF (-18K1) *)
	WY10110_30 AT  %MX10140.30 : BOOL; (*STN 3 ULTRASONIC ON/OFF (-18K1) *)
	WY10110_31 AT  %MX10140.31 : BOOL; (*STN 3 ULTRASONIC ON/OFF (-18K1) *)

	WY10111_00 AT  %MX10144.0 : BOOL; (*STN 1 ELECTRIC ACTUATOR ON/OFF (-21K1) *)
	WY10111_01 AT  %MX10144.1 : BOOL; (*STN 1 ELECTRIC ACTUATOR ON/OFF (-21K1) *)
	WY10111_02 AT  %MX10144.2 : BOOL; (*STN 1 ELECTRIC ACTUATOR ON/OFF (-21K1) *)
	WY10111_03 AT  %MX10144.3 : BOOL; (*STN 1 ELECTRIC ACTUATOR ON/OFF (-21K1) *)
	WY10111_04 AT  %MX10144.4 : BOOL; (*STN 1 ELECTRIC ACTUATOR ON/OFF (-21K1) *)
	WY10111_05 AT  %MX10144.5 : BOOL; (*STN 1 ELECTRIC ACTUATOR ON/OFF (-21K1) *)
	WY10111_06 AT  %MX10144.6 : BOOL; (*STN 1 ELECTRIC ACTUATOR ON/OFF (-21K1) *)
	WY10111_07 AT  %MX10144.7 : BOOL; (*STN 1 ELECTRIC ACTUATOR ON/OFF (-21K1) *)
	WY10111_08 AT  %MX10144.8 : BOOL; (*STN 1 ELECTRIC ACTUATOR ON/OFF (-21K1) *)
	WY10111_09 AT  %MX10144.9 : BOOL; (*STN 1 ELECTRIC ACTUATOR ON/OFF (-21K1) *)
	WY10111_10 AT  %MX10144.10 : BOOL; (*STN 1 ELECTRIC ACTUATOR ON/OFF (-21K1) *)
	WY10111_11 AT  %MX10144.11 : BOOL; (*STN 1 ELECTRIC ACTUATOR ON/OFF (-21K1) *)
	WY10111_12 AT  %MX10144.12 : BOOL; (*STN 1 ELECTRIC ACTUATOR ON/OFF (-21K1) *)
	WY10111_13 AT  %MX10144.13 : BOOL; (*STN 1 ELECTRIC ACTUATOR ON/OFF (-21K1) *)
	WY10111_14 AT  %MX10144.14 : BOOL; (*STN 1 ELECTRIC ACTUATOR ON/OFF (-21K1) *)
	WY10111_15 AT  %MX10144.15 : BOOL; (*STN 1 ELECTRIC ACTUATOR ON/OFF (-21K1) *)
	WY10111_16 AT  %MX10144.16 : BOOL; (*STN 1 ELECTRIC ACTUATOR ON/OFF (-21K1) *)
	WY10111_17 AT  %MX10144.17 : BOOL; (*STN 1 ELECTRIC ACTUATOR ON/OFF (-21K1) *)
	WY10111_18 AT  %MX10144.18 : BOOL; (*STN 1 ELECTRIC ACTUATOR ON/OFF (-21K1) *)
	WY10111_19 AT  %MX10144.19 : BOOL; (*STN 1 ELECTRIC ACTUATOR ON/OFF (-21K1) *)
	WY10111_20 AT  %MX10144.20 : BOOL; (*STN 1 ELECTRIC ACTUATOR ON/OFF (-21K1) *)
	WY10111_21 AT  %MX10144.21 : BOOL; (*STN 1 ELECTRIC ACTUATOR ON/OFF (-21K1) *)
	WY10111_22 AT  %MX10144.22 : BOOL; (*STN 1 ELECTRIC ACTUATOR ON/OFF (-21K1) *)
	WY10111_23 AT  %MX10144.23 : BOOL; (*STN 1 ELECTRIC ACTUATOR ON/OFF (-21K1) *)
	WY10111_24 AT  %MX10144.24 : BOOL; (*STN 1 ELECTRIC ACTUATOR ON/OFF (-21K1) *)
	WY10111_25 AT  %MX10144.25 : BOOL; (*STN 1 ELECTRIC ACTUATOR ON/OFF (-21K1) *)
	WY10111_26 AT  %MX10144.26 : BOOL; (*STN 1 ELECTRIC ACTUATOR ON/OFF (-21K1) *)
	WY10111_27 AT  %MX10144.27 : BOOL; (*STN 1 ELECTRIC ACTUATOR ON/OFF (-21K1) *)
	WY10111_28 AT  %MX10144.28 : BOOL; (*STN 1 ELECTRIC ACTUATOR ON/OFF (-21K1) *)
	WY10111_29 AT  %MX10144.29 : BOOL; (*STN 1 ELECTRIC ACTUATOR ON/OFF (-21K1) *)
	WY10111_30 AT  %MX10144.30 : BOOL; (*STN 1 ELECTRIC ACTUATOR ON/OFF (-21K1) *)
	WY10111_31 AT  %MX10144.31 : BOOL; (*STN 1 ELECTRIC ACTUATOR ON/OFF (-21K1) *)

	WY10112_00 AT  %MX10148.0 : BOOL; (*STN 2 ELECTRIC ACTUATOR ON/OFF (-22K1) *)
	WY10112_01 AT  %MX10148.1 : BOOL; (*STN 2 ELECTRIC ACTUATOR ON/OFF (-22K1) *)
	WY10112_02 AT  %MX10148.2 : BOOL; (*STN 2 ELECTRIC ACTUATOR ON/OFF (-22K1) *)
	WY10112_03 AT  %MX10148.3 : BOOL; (*STN 2 ELECTRIC ACTUATOR ON/OFF (-22K1) *)
	WY10112_04 AT  %MX10148.4 : BOOL; (*STN 2 ELECTRIC ACTUATOR ON/OFF (-22K1) *)
	WY10112_05 AT  %MX10148.5 : BOOL; (*STN 2 ELECTRIC ACTUATOR ON/OFF (-22K1) *)
	WY10112_06 AT  %MX10148.6 : BOOL; (*STN 2 ELECTRIC ACTUATOR ON/OFF (-22K1) *)
	WY10112_07 AT  %MX10148.7 : BOOL; (*STN 2 ELECTRIC ACTUATOR ON/OFF (-22K1) *)
	WY10112_08 AT  %MX10148.8 : BOOL; (*STN 2 ELECTRIC ACTUATOR ON/OFF (-22K1) *)
	WY10112_09 AT  %MX10148.9 : BOOL; (*STN 2 ELECTRIC ACTUATOR ON/OFF (-22K1) *)
	WY10112_10 AT  %MX10148.10 : BOOL; (*STN 2 ELECTRIC ACTUATOR ON/OFF (-22K1) *)
	WY10112_11 AT  %MX10148.11 : BOOL; (*STN 2 ELECTRIC ACTUATOR ON/OFF (-22K1) *)
	WY10112_12 AT  %MX10148.12 : BOOL; (*STN 2 ELECTRIC ACTUATOR ON/OFF (-22K1) *)
	WY10112_13 AT  %MX10148.13 : BOOL; (*STN 2 ELECTRIC ACTUATOR ON/OFF (-22K1) *)
	WY10112_14 AT  %MX10148.14 : BOOL; (*STN 2 ELECTRIC ACTUATOR ON/OFF (-22K1) *)
	WY10112_15 AT  %MX10148.15 : BOOL; (*STN 2 ELECTRIC ACTUATOR ON/OFF (-22K1) *)
	WY10112_16 AT  %MX10148.16 : BOOL; (*STN 2 ELECTRIC ACTUATOR ON/OFF (-22K1) *)
	WY10112_17 AT  %MX10148.17 : BOOL; (*STN 2 ELECTRIC ACTUATOR ON/OFF (-22K1) *)
	WY10112_18 AT  %MX10148.18 : BOOL; (*STN 2 ELECTRIC ACTUATOR ON/OFF (-22K1) *)
	WY10112_19 AT  %MX10148.19 : BOOL; (*STN 2 ELECTRIC ACTUATOR ON/OFF (-22K1) *)
	WY10112_20 AT  %MX10148.20 : BOOL; (*STN 2 ELECTRIC ACTUATOR ON/OFF (-22K1) *)
	WY10112_21 AT  %MX10148.21 : BOOL; (*STN 2 ELECTRIC ACTUATOR ON/OFF (-22K1) *)
	WY10112_22 AT  %MX10148.22 : BOOL; (*STN 2 ELECTRIC ACTUATOR ON/OFF (-22K1) *)
	WY10112_23 AT  %MX10148.23 : BOOL; (*STN 2 ELECTRIC ACTUATOR ON/OFF (-22K1) *)
	WY10112_24 AT  %MX10148.24 : BOOL; (*STN 2 ELECTRIC ACTUATOR ON/OFF (-22K1) *)
	WY10112_25 AT  %MX10148.25 : BOOL; (*STN 2 ELECTRIC ACTUATOR ON/OFF (-22K1) *)
	WY10112_26 AT  %MX10148.26 : BOOL; (*STN 2 ELECTRIC ACTUATOR ON/OFF (-22K1) *)
	WY10112_27 AT  %MX10148.27 : BOOL; (*STN 2 ELECTRIC ACTUATOR ON/OFF (-22K1) *)
	WY10112_28 AT  %MX10148.28 : BOOL; (*STN 2 ELECTRIC ACTUATOR ON/OFF (-22K1) *)
	WY10112_29 AT  %MX10148.29 : BOOL; (*STN 2 ELECTRIC ACTUATOR ON/OFF (-22K1) *)
	WY10112_30 AT  %MX10148.30 : BOOL; (*STN 2 ELECTRIC ACTUATOR ON/OFF (-22K1) *)
	WY10112_31 AT  %MX10148.31 : BOOL; (*STN 2 ELECTRIC ACTUATOR ON/OFF (-22K1) *)

	WY10113_00 AT  %MX10152.0 : BOOL; (*STN 3 ELECTRIC ACTUATOR ON/OFF (-23K1) *)
	WY10113_01 AT  %MX10152.1 : BOOL; (*STN 3 ELECTRIC ACTUATOR ON/OFF (-23K1) *)
	WY10113_02 AT  %MX10152.2 : BOOL; (*STN 3 ELECTRIC ACTUATOR ON/OFF (-23K1) *)
	WY10113_03 AT  %MX10152.3 : BOOL; (*STN 3 ELECTRIC ACTUATOR ON/OFF (-23K1) *)
	WY10113_04 AT  %MX10152.4 : BOOL; (*STN 3 ELECTRIC ACTUATOR ON/OFF (-23K1) *)
	WY10113_05 AT  %MX10152.5 : BOOL; (*STN 3 ELECTRIC ACTUATOR ON/OFF (-23K1) *)
	WY10113_06 AT  %MX10152.6 : BOOL; (*STN 3 ELECTRIC ACTUATOR ON/OFF (-23K1) *)
	WY10113_07 AT  %MX10152.7 : BOOL; (*STN 3 ELECTRIC ACTUATOR ON/OFF (-23K1) *)
	WY10113_08 AT  %MX10152.8 : BOOL; (*STN 3 ELECTRIC ACTUATOR ON/OFF (-23K1) *)
	WY10113_09 AT  %MX10152.9 : BOOL; (*STN 3 ELECTRIC ACTUATOR ON/OFF (-23K1) *)
	WY10113_10 AT  %MX10152.10 : BOOL; (*STN 3 ELECTRIC ACTUATOR ON/OFF (-23K1) *)
	WY10113_11 AT  %MX10152.11 : BOOL; (*STN 3 ELECTRIC ACTUATOR ON/OFF (-23K1) *)
	WY10113_12 AT  %MX10152.12 : BOOL; (*STN 3 ELECTRIC ACTUATOR ON/OFF (-23K1) *)
	WY10113_13 AT  %MX10152.13 : BOOL; (*STN 3 ELECTRIC ACTUATOR ON/OFF (-23K1) *)
	WY10113_14 AT  %MX10152.14 : BOOL; (*STN 3 ELECTRIC ACTUATOR ON/OFF (-23K1) *)
	WY10113_15 AT  %MX10152.15 : BOOL; (*STN 3 ELECTRIC ACTUATOR ON/OFF (-23K1) *)
	WY10113_16 AT  %MX10152.16 : BOOL; (*STN 3 ELECTRIC ACTUATOR ON/OFF (-23K1) *)
	WY10113_17 AT  %MX10152.17 : BOOL; (*STN 3 ELECTRIC ACTUATOR ON/OFF (-23K1) *)
	WY10113_18 AT  %MX10152.18 : BOOL; (*STN 3 ELECTRIC ACTUATOR ON/OFF (-23K1) *)
	WY10113_19 AT  %MX10152.19 : BOOL; (*STN 3 ELECTRIC ACTUATOR ON/OFF (-23K1) *)
	WY10113_20 AT  %MX10152.20 : BOOL; (*STN 3 ELECTRIC ACTUATOR ON/OFF (-23K1) *)
	WY10113_21 AT  %MX10152.21 : BOOL; (*STN 3 ELECTRIC ACTUATOR ON/OFF (-23K1) *)
	WY10113_22 AT  %MX10152.22 : BOOL; (*STN 3 ELECTRIC ACTUATOR ON/OFF (-23K1) *)
	WY10113_23 AT  %MX10152.23 : BOOL; (*STN 3 ELECTRIC ACTUATOR ON/OFF (-23K1) *)
	WY10113_24 AT  %MX10152.24 : BOOL; (*STN 3 ELECTRIC ACTUATOR ON/OFF (-23K1) *)
	WY10113_25 AT  %MX10152.25 : BOOL; (*STN 3 ELECTRIC ACTUATOR ON/OFF (-23K1) *)
	WY10113_26 AT  %MX10152.26 : BOOL; (*STN 3 ELECTRIC ACTUATOR ON/OFF (-23K1) *)
	WY10113_27 AT  %MX10152.27 : BOOL; (*STN 3 ELECTRIC ACTUATOR ON/OFF (-23K1) *)
	WY10113_28 AT  %MX10152.28 : BOOL; (*STN 3 ELECTRIC ACTUATOR ON/OFF (-23K1) *)
	WY10113_29 AT  %MX10152.29 : BOOL; (*STN 3 ELECTRIC ACTUATOR ON/OFF (-23K1) *)
	WY10113_30 AT  %MX10152.30 : BOOL; (*STN 3 ELECTRIC ACTUATOR ON/OFF (-23K1) *)
	WY10113_31 AT  %MX10152.31 : BOOL; (*STN 3 ELECTRIC ACTUATOR ON/OFF (-23K1) *)

	WY10114_00 AT  %MX10156.0 : BOOL; (*RESERVED *)
	WY10114_01 AT  %MX10156.1 : BOOL; (*RESERVED *)
	WY10114_02 AT  %MX10156.2 : BOOL; (*RESERVED *)
	WY10114_03 AT  %MX10156.3 : BOOL; (*RESERVED *)
	WY10114_04 AT  %MX10156.4 : BOOL; (*RESERVED *)
	WY10114_05 AT  %MX10156.5 : BOOL; (*RESERVED *)
	WY10114_06 AT  %MX10156.6 : BOOL; (*RESERVED *)
	WY10114_07 AT  %MX10156.7 : BOOL; (*RESERVED *)
	WY10114_08 AT  %MX10156.8 : BOOL; (*RESERVED *)
	WY10114_09 AT  %MX10156.9 : BOOL; (*RESERVED *)
	WY10114_10 AT  %MX10156.10 : BOOL; (*RESERVED *)
	WY10114_11 AT  %MX10156.11 : BOOL; (*RESERVED *)
	WY10114_12 AT  %MX10156.12 : BOOL; (*RESERVED *)
	WY10114_13 AT  %MX10156.13 : BOOL; (*RESERVED *)
	WY10114_14 AT  %MX10156.14 : BOOL; (*RESERVED *)
	WY10114_15 AT  %MX10156.15 : BOOL; (*RESERVED *)
	WY10114_16 AT  %MX10156.16 : BOOL; (*RESERVED *)
	WY10114_17 AT  %MX10156.17 : BOOL; (*RESERVED *)
	WY10114_18 AT  %MX10156.18 : BOOL; (*RESERVED *)
	WY10114_19 AT  %MX10156.19 : BOOL; (*RESERVED *)
	WY10114_20 AT  %MX10156.20 : BOOL; (*RESERVED *)
	WY10114_21 AT  %MX10156.21 : BOOL; (*RESERVED *)
	WY10114_22 AT  %MX10156.22 : BOOL; (*RESERVED *)
	WY10114_23 AT  %MX10156.23 : BOOL; (*RESERVED *)
	WY10114_24 AT  %MX10156.24 : BOOL; (*RESERVED *)
	WY10114_25 AT  %MX10156.25 : BOOL; (*RESERVED *)
	WY10114_26 AT  %MX10156.26 : BOOL; (*RESERVED *)
	WY10114_27 AT  %MX10156.27 : BOOL; (*RESERVED *)
	WY10114_28 AT  %MX10156.28 : BOOL; (*RESERVED *)
	WY10114_29 AT  %MX10156.29 : BOOL; (*RESERVED *)
	WY10114_30 AT  %MX10156.30 : BOOL; (*RESERVED *)
	WY10114_31 AT  %MX10156.31 : BOOL; (*RESERVED *)

	WY10115_00 AT  %MX10160.0 : BOOL; (*RESERVED *)
	WY10115_01 AT  %MX10160.1 : BOOL; (*RESERVED *)
	WY10115_02 AT  %MX10160.2 : BOOL; (*RESERVED *)
	WY10115_03 AT  %MX10160.3 : BOOL; (*RESERVED *)
	WY10115_04 AT  %MX10160.4 : BOOL; (*RESERVED *)
	WY10115_05 AT  %MX10160.5 : BOOL; (*RESERVED *)
	WY10115_06 AT  %MX10160.6 : BOOL; (*RESERVED *)
	WY10115_07 AT  %MX10160.7 : BOOL; (*RESERVED *)
	WY10115_08 AT  %MX10160.8 : BOOL; (*RESERVED *)
	WY10115_09 AT  %MX10160.9 : BOOL; (*RESERVED *)
	WY10115_10 AT  %MX10160.10 : BOOL; (*RESERVED *)
	WY10115_11 AT  %MX10160.11 : BOOL; (*RESERVED *)
	WY10115_12 AT  %MX10160.12 : BOOL; (*RESERVED *)
	WY10115_13 AT  %MX10160.13 : BOOL; (*RESERVED *)
	WY10115_14 AT  %MX10160.14 : BOOL; (*RESERVED *)
	WY10115_15 AT  %MX10160.15 : BOOL; (*RESERVED *)
	WY10115_16 AT  %MX10160.16 : BOOL; (*RESERVED *)
	WY10115_17 AT  %MX10160.17 : BOOL; (*RESERVED *)
	WY10115_18 AT  %MX10160.18 : BOOL; (*RESERVED *)
	WY10115_19 AT  %MX10160.19 : BOOL; (*RESERVED *)
	WY10115_20 AT  %MX10160.20 : BOOL; (*RESERVED *)
	WY10115_21 AT  %MX10160.21 : BOOL; (*RESERVED *)
	WY10115_22 AT  %MX10160.22 : BOOL; (*RESERVED *)
	WY10115_23 AT  %MX10160.23 : BOOL; (*RESERVED *)
	WY10115_24 AT  %MX10160.24 : BOOL; (*RESERVED *)
	WY10115_25 AT  %MX10160.25 : BOOL; (*RESERVED *)
	WY10115_26 AT  %MX10160.26 : BOOL; (*RESERVED *)
	WY10115_27 AT  %MX10160.27 : BOOL; (*RESERVED *)
	WY10115_28 AT  %MX10160.28 : BOOL; (*RESERVED *)
	WY10115_29 AT  %MX10160.29 : BOOL; (*RESERVED *)
	WY10115_30 AT  %MX10160.30 : BOOL; (*RESERVED *)
	WY10115_31 AT  %MX10160.31 : BOOL; (*RESERVED *)

	WY10200_00 AT  %MX10200.0 : BOOL; (*STN 5 PROCESS TANK HEATER A ON/OFF (-70K1) *)
	WY10200_01 AT  %MX10200.1 : BOOL; (*STN 5 PROCESS TANK HEATER A ON/OFF (-70K1) *)
	WY10200_02 AT  %MX10200.2 : BOOL; (*STN 5 PROCESS TANK HEATER A ON/OFF (-70K1) *)
	WY10200_03 AT  %MX10200.3 : BOOL; (*STN 5 PROCESS TANK HEATER A ON/OFF (-70K1) *)
	WY10200_04 AT  %MX10200.4 : BOOL; (*STN 5 PROCESS TANK HEATER A ON/OFF (-70K1) *)
	WY10200_05 AT  %MX10200.5 : BOOL; (*STN 5 PROCESS TANK HEATER A ON/OFF (-70K1) *)
	WY10200_06 AT  %MX10200.6 : BOOL; (*STN 5 PROCESS TANK HEATER A ON/OFF (-70K1) *)
	WY10200_07 AT  %MX10200.7 : BOOL; (*STN 5 PROCESS TANK HEATER A ON/OFF (-70K1) *)
	WY10200_08 AT  %MX10200.8 : BOOL; (*STN 5 PROCESS TANK HEATER A ON/OFF (-70K1) *)
	WY10200_09 AT  %MX10200.9 : BOOL; (*STN 5 PROCESS TANK HEATER A ON/OFF (-70K1) *)
	WY10200_10 AT  %MX10200.10 : BOOL; (*STN 5 PROCESS TANK HEATER A ON/OFF (-70K1) *)
	WY10200_11 AT  %MX10200.11 : BOOL; (*STN 5 PROCESS TANK HEATER A ON/OFF (-70K1) *)
	WY10200_12 AT  %MX10200.12 : BOOL; (*STN 5 PROCESS TANK HEATER A ON/OFF (-70K1) *)
	WY10200_13 AT  %MX10200.13 : BOOL; (*STN 5 PROCESS TANK HEATER A ON/OFF (-70K1) *)
	WY10200_14 AT  %MX10200.14 : BOOL; (*STN 5 PROCESS TANK HEATER A ON/OFF (-70K1) *)
	WY10200_15 AT  %MX10200.15 : BOOL; (*STN 5 PROCESS TANK HEATER A ON/OFF (-70K1) *)
	WY10200_16 AT  %MX10200.16 : BOOL; (*STN 5 PROCESS TANK HEATER A ON/OFF (-70K1) *)
	WY10200_17 AT  %MX10200.17 : BOOL; (*STN 5 PROCESS TANK HEATER A ON/OFF (-70K1) *)
	WY10200_18 AT  %MX10200.18 : BOOL; (*STN 5 PROCESS TANK HEATER A ON/OFF (-70K1) *)
	WY10200_19 AT  %MX10200.19 : BOOL; (*STN 5 PROCESS TANK HEATER A ON/OFF (-70K1) *)
	WY10200_20 AT  %MX10200.20 : BOOL; (*STN 5 PROCESS TANK HEATER A ON/OFF (-70K1) *)
	WY10200_21 AT  %MX10200.21 : BOOL; (*STN 5 PROCESS TANK HEATER A ON/OFF (-70K1) *)
	WY10200_22 AT  %MX10200.22 : BOOL; (*STN 5 PROCESS TANK HEATER A ON/OFF (-70K1) *)
	WY10200_23 AT  %MX10200.23 : BOOL; (*STN 5 PROCESS TANK HEATER A ON/OFF (-70K1) *)
	WY10200_24 AT  %MX10200.24 : BOOL; (*STN 5 PROCESS TANK HEATER A ON/OFF (-70K1) *)
	WY10200_25 AT  %MX10200.25 : BOOL; (*STN 5 PROCESS TANK HEATER A ON/OFF (-70K1) *)
	WY10200_26 AT  %MX10200.26 : BOOL; (*STN 5 PROCESS TANK HEATER A ON/OFF (-70K1) *)
	WY10200_27 AT  %MX10200.27 : BOOL; (*STN 5 PROCESS TANK HEATER A ON/OFF (-70K1) *)
	WY10200_28 AT  %MX10200.28 : BOOL; (*STN 5 PROCESS TANK HEATER A ON/OFF (-70K1) *)
	WY10200_29 AT  %MX10200.29 : BOOL; (*STN 5 PROCESS TANK HEATER A ON/OFF (-70K1) *)
	WY10200_30 AT  %MX10200.30 : BOOL; (*STN 5 PROCESS TANK HEATER A ON/OFF (-70K1) *)
	WY10200_31 AT  %MX10200.31 : BOOL; (*STN 5 PROCESS TANK HEATER A ON/OFF (-70K1) *)

	WY10201_00 AT  %MX10204.0 : BOOL; (*STN 5 PROCESS TANK HEATER B ON/OFF (-71K1) *)
	WY10201_01 AT  %MX10204.1 : BOOL; (*STN 5 PROCESS TANK HEATER B ON/OFF (-71K1) *)
	WY10201_02 AT  %MX10204.2 : BOOL; (*STN 5 PROCESS TANK HEATER B ON/OFF (-71K1) *)
	WY10201_03 AT  %MX10204.3 : BOOL; (*STN 5 PROCESS TANK HEATER B ON/OFF (-71K1) *)
	WY10201_04 AT  %MX10204.4 : BOOL; (*STN 5 PROCESS TANK HEATER B ON/OFF (-71K1) *)
	WY10201_05 AT  %MX10204.5 : BOOL; (*STN 5 PROCESS TANK HEATER B ON/OFF (-71K1) *)
	WY10201_06 AT  %MX10204.6 : BOOL; (*STN 5 PROCESS TANK HEATER B ON/OFF (-71K1) *)
	WY10201_07 AT  %MX10204.7 : BOOL; (*STN 5 PROCESS TANK HEATER B ON/OFF (-71K1) *)
	WY10201_08 AT  %MX10204.8 : BOOL; (*STN 5 PROCESS TANK HEATER B ON/OFF (-71K1) *)
	WY10201_09 AT  %MX10204.9 : BOOL; (*STN 5 PROCESS TANK HEATER B ON/OFF (-71K1) *)
	WY10201_10 AT  %MX10204.10 : BOOL; (*STN 5 PROCESS TANK HEATER B ON/OFF (-71K1) *)
	WY10201_11 AT  %MX10204.11 : BOOL; (*STN 5 PROCESS TANK HEATER B ON/OFF (-71K1) *)
	WY10201_12 AT  %MX10204.12 : BOOL; (*STN 5 PROCESS TANK HEATER B ON/OFF (-71K1) *)
	WY10201_13 AT  %MX10204.13 : BOOL; (*STN 5 PROCESS TANK HEATER B ON/OFF (-71K1) *)
	WY10201_14 AT  %MX10204.14 : BOOL; (*STN 5 PROCESS TANK HEATER B ON/OFF (-71K1) *)
	WY10201_15 AT  %MX10204.15 : BOOL; (*STN 5 PROCESS TANK HEATER B ON/OFF (-71K1) *)
	WY10201_16 AT  %MX10204.16 : BOOL; (*STN 5 PROCESS TANK HEATER B ON/OFF (-71K1) *)
	WY10201_17 AT  %MX10204.17 : BOOL; (*STN 5 PROCESS TANK HEATER B ON/OFF (-71K1) *)
	WY10201_18 AT  %MX10204.18 : BOOL; (*STN 5 PROCESS TANK HEATER B ON/OFF (-71K1) *)
	WY10201_19 AT  %MX10204.19 : BOOL; (*STN 5 PROCESS TANK HEATER B ON/OFF (-71K1) *)
	WY10201_20 AT  %MX10204.20 : BOOL; (*STN 5 PROCESS TANK HEATER B ON/OFF (-71K1) *)
	WY10201_21 AT  %MX10204.21 : BOOL; (*STN 5 PROCESS TANK HEATER B ON/OFF (-71K1) *)
	WY10201_22 AT  %MX10204.22 : BOOL; (*STN 5 PROCESS TANK HEATER B ON/OFF (-71K1) *)
	WY10201_23 AT  %MX10204.23 : BOOL; (*STN 5 PROCESS TANK HEATER B ON/OFF (-71K1) *)
	WY10201_24 AT  %MX10204.24 : BOOL; (*STN 5 PROCESS TANK HEATER B ON/OFF (-71K1) *)
	WY10201_25 AT  %MX10204.25 : BOOL; (*STN 5 PROCESS TANK HEATER B ON/OFF (-71K1) *)
	WY10201_26 AT  %MX10204.26 : BOOL; (*STN 5 PROCESS TANK HEATER B ON/OFF (-71K1) *)
	WY10201_27 AT  %MX10204.27 : BOOL; (*STN 5 PROCESS TANK HEATER B ON/OFF (-71K1) *)
	WY10201_28 AT  %MX10204.28 : BOOL; (*STN 5 PROCESS TANK HEATER B ON/OFF (-71K1) *)
	WY10201_29 AT  %MX10204.29 : BOOL; (*STN 5 PROCESS TANK HEATER B ON/OFF (-71K1) *)
	WY10201_30 AT  %MX10204.30 : BOOL; (*STN 5 PROCESS TANK HEATER B ON/OFF (-71K1) *)
	WY10201_31 AT  %MX10204.31 : BOOL; (*STN 5 PROCESS TANK HEATER B ON/OFF (-71K1) *)

	WY10202_00 AT  %MX10208.0 : BOOL; (*STN 1 SUB PROCESS TANK HEATER ON/OFF (-72K1) *)
	WY10202_01 AT  %MX10208.1 : BOOL; (*STN 1 SUB PROCESS TANK HEATER ON/OFF (-72K1) *)
	WY10202_02 AT  %MX10208.2 : BOOL; (*STN 1 SUB PROCESS TANK HEATER ON/OFF (-72K1) *)
	WY10202_03 AT  %MX10208.3 : BOOL; (*STN 1 SUB PROCESS TANK HEATER ON/OFF (-72K1) *)
	WY10202_04 AT  %MX10208.4 : BOOL; (*STN 1 SUB PROCESS TANK HEATER ON/OFF (-72K1) *)
	WY10202_05 AT  %MX10208.5 : BOOL; (*STN 1 SUB PROCESS TANK HEATER ON/OFF (-72K1) *)
	WY10202_06 AT  %MX10208.6 : BOOL; (*STN 1 SUB PROCESS TANK HEATER ON/OFF (-72K1) *)
	WY10202_07 AT  %MX10208.7 : BOOL; (*STN 1 SUB PROCESS TANK HEATER ON/OFF (-72K1) *)
	WY10202_08 AT  %MX10208.8 : BOOL; (*STN 1 SUB PROCESS TANK HEATER ON/OFF (-72K1) *)
	WY10202_09 AT  %MX10208.9 : BOOL; (*STN 1 SUB PROCESS TANK HEATER ON/OFF (-72K1) *)
	WY10202_10 AT  %MX10208.10 : BOOL; (*STN 1 SUB PROCESS TANK HEATER ON/OFF (-72K1) *)
	WY10202_11 AT  %MX10208.11 : BOOL; (*STN 1 SUB PROCESS TANK HEATER ON/OFF (-72K1) *)
	WY10202_12 AT  %MX10208.12 : BOOL; (*STN 1 SUB PROCESS TANK HEATER ON/OFF (-72K1) *)
	WY10202_13 AT  %MX10208.13 : BOOL; (*STN 1 SUB PROCESS TANK HEATER ON/OFF (-72K1) *)
	WY10202_14 AT  %MX10208.14 : BOOL; (*STN 1 SUB PROCESS TANK HEATER ON/OFF (-72K1) *)
	WY10202_15 AT  %MX10208.15 : BOOL; (*STN 1 SUB PROCESS TANK HEATER ON/OFF (-72K1) *)
	WY10202_16 AT  %MX10208.16 : BOOL; (*STN 1 SUB PROCESS TANK HEATER ON/OFF (-72K1) *)
	WY10202_17 AT  %MX10208.17 : BOOL; (*STN 1 SUB PROCESS TANK HEATER ON/OFF (-72K1) *)
	WY10202_18 AT  %MX10208.18 : BOOL; (*STN 1 SUB PROCESS TANK HEATER ON/OFF (-72K1) *)
	WY10202_19 AT  %MX10208.19 : BOOL; (*STN 1 SUB PROCESS TANK HEATER ON/OFF (-72K1) *)
	WY10202_20 AT  %MX10208.20 : BOOL; (*STN 1 SUB PROCESS TANK HEATER ON/OFF (-72K1) *)
	WY10202_21 AT  %MX10208.21 : BOOL; (*STN 1 SUB PROCESS TANK HEATER ON/OFF (-72K1) *)
	WY10202_22 AT  %MX10208.22 : BOOL; (*STN 1 SUB PROCESS TANK HEATER ON/OFF (-72K1) *)
	WY10202_23 AT  %MX10208.23 : BOOL; (*STN 1 SUB PROCESS TANK HEATER ON/OFF (-72K1) *)
	WY10202_24 AT  %MX10208.24 : BOOL; (*STN 1 SUB PROCESS TANK HEATER ON/OFF (-72K1) *)
	WY10202_25 AT  %MX10208.25 : BOOL; (*STN 1 SUB PROCESS TANK HEATER ON/OFF (-72K1) *)
	WY10202_26 AT  %MX10208.26 : BOOL; (*STN 1 SUB PROCESS TANK HEATER ON/OFF (-72K1) *)
	WY10202_27 AT  %MX10208.27 : BOOL; (*STN 1 SUB PROCESS TANK HEATER ON/OFF (-72K1) *)
	WY10202_28 AT  %MX10208.28 : BOOL; (*STN 1 SUB PROCESS TANK HEATER ON/OFF (-72K1) *)
	WY10202_29 AT  %MX10208.29 : BOOL; (*STN 1 SUB PROCESS TANK HEATER ON/OFF (-72K1) *)
	WY10202_30 AT  %MX10208.30 : BOOL; (*STN 1 SUB PROCESS TANK HEATER ON/OFF (-72K1) *)
	WY10202_31 AT  %MX10208.31 : BOOL; (*STN 1 SUB PROCESS TANK HEATER ON/OFF (-72K1) *)

	WY10203_00 AT  %MX10212.0 : BOOL; (*STN 2 SUB PROCESS TANK HEATER ON/OFF (-73K1) *)
	WY10203_01 AT  %MX10212.1 : BOOL; (*STN 2 SUB PROCESS TANK HEATER ON/OFF (-73K1) *)
	WY10203_02 AT  %MX10212.2 : BOOL; (*STN 2 SUB PROCESS TANK HEATER ON/OFF (-73K1) *)
	WY10203_03 AT  %MX10212.3 : BOOL; (*STN 2 SUB PROCESS TANK HEATER ON/OFF (-73K1) *)
	WY10203_04 AT  %MX10212.4 : BOOL; (*STN 2 SUB PROCESS TANK HEATER ON/OFF (-73K1) *)
	WY10203_05 AT  %MX10212.5 : BOOL; (*STN 2 SUB PROCESS TANK HEATER ON/OFF (-73K1) *)
	WY10203_06 AT  %MX10212.6 : BOOL; (*STN 2 SUB PROCESS TANK HEATER ON/OFF (-73K1) *)
	WY10203_07 AT  %MX10212.7 : BOOL; (*STN 2 SUB PROCESS TANK HEATER ON/OFF (-73K1) *)
	WY10203_08 AT  %MX10212.8 : BOOL; (*STN 2 SUB PROCESS TANK HEATER ON/OFF (-73K1) *)
	WY10203_09 AT  %MX10212.9 : BOOL; (*STN 2 SUB PROCESS TANK HEATER ON/OFF (-73K1) *)
	WY10203_10 AT  %MX10212.10 : BOOL; (*STN 2 SUB PROCESS TANK HEATER ON/OFF (-73K1) *)
	WY10203_11 AT  %MX10212.11 : BOOL; (*STN 2 SUB PROCESS TANK HEATER ON/OFF (-73K1) *)
	WY10203_12 AT  %MX10212.12 : BOOL; (*STN 2 SUB PROCESS TANK HEATER ON/OFF (-73K1) *)
	WY10203_13 AT  %MX10212.13 : BOOL; (*STN 2 SUB PROCESS TANK HEATER ON/OFF (-73K1) *)
	WY10203_14 AT  %MX10212.14 : BOOL; (*STN 2 SUB PROCESS TANK HEATER ON/OFF (-73K1) *)
	WY10203_15 AT  %MX10212.15 : BOOL; (*STN 2 SUB PROCESS TANK HEATER ON/OFF (-73K1) *)
	WY10203_16 AT  %MX10212.16 : BOOL; (*STN 2 SUB PROCESS TANK HEATER ON/OFF (-73K1) *)
	WY10203_17 AT  %MX10212.17 : BOOL; (*STN 2 SUB PROCESS TANK HEATER ON/OFF (-73K1) *)
	WY10203_18 AT  %MX10212.18 : BOOL; (*STN 2 SUB PROCESS TANK HEATER ON/OFF (-73K1) *)
	WY10203_19 AT  %MX10212.19 : BOOL; (*STN 2 SUB PROCESS TANK HEATER ON/OFF (-73K1) *)
	WY10203_20 AT  %MX10212.20 : BOOL; (*STN 2 SUB PROCESS TANK HEATER ON/OFF (-73K1) *)
	WY10203_21 AT  %MX10212.21 : BOOL; (*STN 2 SUB PROCESS TANK HEATER ON/OFF (-73K1) *)
	WY10203_22 AT  %MX10212.22 : BOOL; (*STN 2 SUB PROCESS TANK HEATER ON/OFF (-73K1) *)
	WY10203_23 AT  %MX10212.23 : BOOL; (*STN 2 SUB PROCESS TANK HEATER ON/OFF (-73K1) *)
	WY10203_24 AT  %MX10212.24 : BOOL; (*STN 2 SUB PROCESS TANK HEATER ON/OFF (-73K1) *)
	WY10203_25 AT  %MX10212.25 : BOOL; (*STN 2 SUB PROCESS TANK HEATER ON/OFF (-73K1) *)
	WY10203_26 AT  %MX10212.26 : BOOL; (*STN 2 SUB PROCESS TANK HEATER ON/OFF (-73K1) *)
	WY10203_27 AT  %MX10212.27 : BOOL; (*STN 2 SUB PROCESS TANK HEATER ON/OFF (-73K1) *)
	WY10203_28 AT  %MX10212.28 : BOOL; (*STN 2 SUB PROCESS TANK HEATER ON/OFF (-73K1) *)
	WY10203_29 AT  %MX10212.29 : BOOL; (*STN 2 SUB PROCESS TANK HEATER ON/OFF (-73K1) *)
	WY10203_30 AT  %MX10212.30 : BOOL; (*STN 2 SUB PROCESS TANK HEATER ON/OFF (-73K1) *)
	WY10203_31 AT  %MX10212.31 : BOOL; (*STN 2 SUB PROCESS TANK HEATER ON/OFF (-73K1) *)

	WY10204_00 AT  %MX10216.0 : BOOL; (*STN 3 SUB PROCESS TANK HEATER ON/OFF (-74K1) *)
	WY10204_01 AT  %MX10216.1 : BOOL; (*STN 3 SUB PROCESS TANK HEATER ON/OFF (-74K1) *)
	WY10204_02 AT  %MX10216.2 : BOOL; (*STN 3 SUB PROCESS TANK HEATER ON/OFF (-74K1) *)
	WY10204_03 AT  %MX10216.3 : BOOL; (*STN 3 SUB PROCESS TANK HEATER ON/OFF (-74K1) *)
	WY10204_04 AT  %MX10216.4 : BOOL; (*STN 3 SUB PROCESS TANK HEATER ON/OFF (-74K1) *)
	WY10204_05 AT  %MX10216.5 : BOOL; (*STN 3 SUB PROCESS TANK HEATER ON/OFF (-74K1) *)
	WY10204_06 AT  %MX10216.6 : BOOL; (*STN 3 SUB PROCESS TANK HEATER ON/OFF (-74K1) *)
	WY10204_07 AT  %MX10216.7 : BOOL; (*STN 3 SUB PROCESS TANK HEATER ON/OFF (-74K1) *)
	WY10204_08 AT  %MX10216.8 : BOOL; (*STN 3 SUB PROCESS TANK HEATER ON/OFF (-74K1) *)
	WY10204_09 AT  %MX10216.9 : BOOL; (*STN 3 SUB PROCESS TANK HEATER ON/OFF (-74K1) *)
	WY10204_10 AT  %MX10216.10 : BOOL; (*STN 3 SUB PROCESS TANK HEATER ON/OFF (-74K1) *)
	WY10204_11 AT  %MX10216.11 : BOOL; (*STN 3 SUB PROCESS TANK HEATER ON/OFF (-74K1) *)
	WY10204_12 AT  %MX10216.12 : BOOL; (*STN 3 SUB PROCESS TANK HEATER ON/OFF (-74K1) *)
	WY10204_13 AT  %MX10216.13 : BOOL; (*STN 3 SUB PROCESS TANK HEATER ON/OFF (-74K1) *)
	WY10204_14 AT  %MX10216.14 : BOOL; (*STN 3 SUB PROCESS TANK HEATER ON/OFF (-74K1) *)
	WY10204_15 AT  %MX10216.15 : BOOL; (*STN 3 SUB PROCESS TANK HEATER ON/OFF (-74K1) *)
	WY10204_16 AT  %MX10216.16 : BOOL; (*STN 3 SUB PROCESS TANK HEATER ON/OFF (-74K1) *)
	WY10204_17 AT  %MX10216.17 : BOOL; (*STN 3 SUB PROCESS TANK HEATER ON/OFF (-74K1) *)
	WY10204_18 AT  %MX10216.18 : BOOL; (*STN 3 SUB PROCESS TANK HEATER ON/OFF (-74K1) *)
	WY10204_19 AT  %MX10216.19 : BOOL; (*STN 3 SUB PROCESS TANK HEATER ON/OFF (-74K1) *)
	WY10204_20 AT  %MX10216.20 : BOOL; (*STN 3 SUB PROCESS TANK HEATER ON/OFF (-74K1) *)
	WY10204_21 AT  %MX10216.21 : BOOL; (*STN 3 SUB PROCESS TANK HEATER ON/OFF (-74K1) *)
	WY10204_22 AT  %MX10216.22 : BOOL; (*STN 3 SUB PROCESS TANK HEATER ON/OFF (-74K1) *)
	WY10204_23 AT  %MX10216.23 : BOOL; (*STN 3 SUB PROCESS TANK HEATER ON/OFF (-74K1) *)
	WY10204_24 AT  %MX10216.24 : BOOL; (*STN 3 SUB PROCESS TANK HEATER ON/OFF (-74K1) *)
	WY10204_25 AT  %MX10216.25 : BOOL; (*STN 3 SUB PROCESS TANK HEATER ON/OFF (-74K1) *)
	WY10204_26 AT  %MX10216.26 : BOOL; (*STN 3 SUB PROCESS TANK HEATER ON/OFF (-74K1) *)
	WY10204_27 AT  %MX10216.27 : BOOL; (*STN 3 SUB PROCESS TANK HEATER ON/OFF (-74K1) *)
	WY10204_28 AT  %MX10216.28 : BOOL; (*STN 3 SUB PROCESS TANK HEATER ON/OFF (-74K1) *)
	WY10204_29 AT  %MX10216.29 : BOOL; (*STN 3 SUB PROCESS TANK HEATER ON/OFF (-74K1) *)
	WY10204_30 AT  %MX10216.30 : BOOL; (*STN 3 SUB PROCESS TANK HEATER ON/OFF (-74K1) *)
	WY10204_31 AT  %MX10216.31 : BOOL; (*STN 3 SUB PROCESS TANK HEATER ON/OFF (-74K1) *)

	WY10205_00 AT  %MX10220.0 : BOOL; (*MAIN INC HEATER ON/OFF   (-75K1) *)
	WY10205_01 AT  %MX10220.1 : BOOL; (*MAIN INC HEATER ON/OFF   (-75K1) *)
	WY10205_02 AT  %MX10220.2 : BOOL; (*MAIN INC HEATER ON/OFF   (-75K1) *)
	WY10205_03 AT  %MX10220.3 : BOOL; (*MAIN INC HEATER ON/OFF   (-75K1) *)
	WY10205_04 AT  %MX10220.4 : BOOL; (*MAIN INC HEATER ON/OFF   (-75K1) *)
	WY10205_05 AT  %MX10220.5 : BOOL; (*MAIN INC HEATER ON/OFF   (-75K1) *)
	WY10205_06 AT  %MX10220.6 : BOOL; (*MAIN INC HEATER ON/OFF   (-75K1) *)
	WY10205_07 AT  %MX10220.7 : BOOL; (*MAIN INC HEATER ON/OFF   (-75K1) *)
	WY10205_08 AT  %MX10220.8 : BOOL; (*MAIN INC HEATER ON/OFF   (-75K1) *)
	WY10205_09 AT  %MX10220.9 : BOOL; (*MAIN INC HEATER ON/OFF   (-75K1) *)
	WY10205_10 AT  %MX10220.10 : BOOL; (*MAIN INC HEATER ON/OFF   (-75K1) *)
	WY10205_11 AT  %MX10220.11 : BOOL; (*MAIN INC HEATER ON/OFF   (-75K1) *)
	WY10205_12 AT  %MX10220.12 : BOOL; (*MAIN INC HEATER ON/OFF   (-75K1) *)
	WY10205_13 AT  %MX10220.13 : BOOL; (*MAIN INC HEATER ON/OFF   (-75K1) *)
	WY10205_14 AT  %MX10220.14 : BOOL; (*MAIN INC HEATER ON/OFF   (-75K1) *)
	WY10205_15 AT  %MX10220.15 : BOOL; (*MAIN INC HEATER ON/OFF   (-75K1) *)
	WY10205_16 AT  %MX10220.16 : BOOL; (*MAIN INC HEATER ON/OFF   (-75K1) *)
	WY10205_17 AT  %MX10220.17 : BOOL; (*MAIN INC HEATER ON/OFF   (-75K1) *)
	WY10205_18 AT  %MX10220.18 : BOOL; (*MAIN INC HEATER ON/OFF   (-75K1) *)
	WY10205_19 AT  %MX10220.19 : BOOL; (*MAIN INC HEATER ON/OFF   (-75K1) *)
	WY10205_20 AT  %MX10220.20 : BOOL; (*MAIN INC HEATER ON/OFF   (-75K1) *)
	WY10205_21 AT  %MX10220.21 : BOOL; (*MAIN INC HEATER ON/OFF   (-75K1) *)
	WY10205_22 AT  %MX10220.22 : BOOL; (*MAIN INC HEATER ON/OFF   (-75K1) *)
	WY10205_23 AT  %MX10220.23 : BOOL; (*MAIN INC HEATER ON/OFF   (-75K1) *)
	WY10205_24 AT  %MX10220.24 : BOOL; (*MAIN INC HEATER ON/OFF   (-75K1) *)
	WY10205_25 AT  %MX10220.25 : BOOL; (*MAIN INC HEATER ON/OFF   (-75K1) *)
	WY10205_26 AT  %MX10220.26 : BOOL; (*MAIN INC HEATER ON/OFF   (-75K1) *)
	WY10205_27 AT  %MX10220.27 : BOOL; (*MAIN INC HEATER ON/OFF   (-75K1) *)
	WY10205_28 AT  %MX10220.28 : BOOL; (*MAIN INC HEATER ON/OFF   (-75K1) *)
	WY10205_29 AT  %MX10220.29 : BOOL; (*MAIN INC HEATER ON/OFF   (-75K1) *)
	WY10205_30 AT  %MX10220.30 : BOOL; (*MAIN INC HEATER ON/OFF   (-75K1) *)
	WY10205_31 AT  %MX10220.31 : BOOL; (*MAIN INC HEATER ON/OFF   (-75K1) *)

	WY10206_00 AT  %MX10224.0 : BOOL; (*STN 1 ULTRASONIC FREQ ON/OFF (-16U1) *)
	WY10206_01 AT  %MX10224.1 : BOOL; (*STN 1 ULTRASONIC FREQ ON/OFF (-16U1) *)
	WY10206_02 AT  %MX10224.2 : BOOL; (*STN 1 ULTRASONIC FREQ ON/OFF (-16U1) *)
	WY10206_03 AT  %MX10224.3 : BOOL; (*STN 1 ULTRASONIC FREQ ON/OFF (-16U1) *)
	WY10206_04 AT  %MX10224.4 : BOOL; (*STN 1 ULTRASONIC FREQ ON/OFF (-16U1) *)
	WY10206_05 AT  %MX10224.5 : BOOL; (*STN 1 ULTRASONIC FREQ ON/OFF (-16U1) *)
	WY10206_06 AT  %MX10224.6 : BOOL; (*STN 1 ULTRASONIC FREQ ON/OFF (-16U1) *)
	WY10206_07 AT  %MX10224.7 : BOOL; (*STN 1 ULTRASONIC FREQ ON/OFF (-16U1) *)
	WY10206_08 AT  %MX10224.8 : BOOL; (*STN 1 ULTRASONIC FREQ ON/OFF (-16U1) *)
	WY10206_09 AT  %MX10224.9 : BOOL; (*STN 1 ULTRASONIC FREQ ON/OFF (-16U1) *)
	WY10206_10 AT  %MX10224.10 : BOOL; (*STN 1 ULTRASONIC FREQ ON/OFF (-16U1) *)
	WY10206_11 AT  %MX10224.11 : BOOL; (*STN 1 ULTRASONIC FREQ ON/OFF (-16U1) *)
	WY10206_12 AT  %MX10224.12 : BOOL; (*STN 1 ULTRASONIC FREQ ON/OFF (-16U1) *)
	WY10206_13 AT  %MX10224.13 : BOOL; (*STN 1 ULTRASONIC FREQ ON/OFF (-16U1) *)
	WY10206_14 AT  %MX10224.14 : BOOL; (*STN 1 ULTRASONIC FREQ ON/OFF (-16U1) *)
	WY10206_15 AT  %MX10224.15 : BOOL; (*STN 1 ULTRASONIC FREQ ON/OFF (-16U1) *)
	WY10206_16 AT  %MX10224.16 : BOOL; (*STN 1 ULTRASONIC FREQ ON/OFF (-16U1) *)
	WY10206_17 AT  %MX10224.17 : BOOL; (*STN 1 ULTRASONIC FREQ ON/OFF (-16U1) *)
	WY10206_18 AT  %MX10224.18 : BOOL; (*STN 1 ULTRASONIC FREQ ON/OFF (-16U1) *)
	WY10206_19 AT  %MX10224.19 : BOOL; (*STN 1 ULTRASONIC FREQ ON/OFF (-16U1) *)
	WY10206_20 AT  %MX10224.20 : BOOL; (*STN 1 ULTRASONIC FREQ ON/OFF (-16U1) *)
	WY10206_21 AT  %MX10224.21 : BOOL; (*STN 1 ULTRASONIC FREQ ON/OFF (-16U1) *)
	WY10206_22 AT  %MX10224.22 : BOOL; (*STN 1 ULTRASONIC FREQ ON/OFF (-16U1) *)
	WY10206_23 AT  %MX10224.23 : BOOL; (*STN 1 ULTRASONIC FREQ ON/OFF (-16U1) *)
	WY10206_24 AT  %MX10224.24 : BOOL; (*STN 1 ULTRASONIC FREQ ON/OFF (-16U1) *)
	WY10206_25 AT  %MX10224.25 : BOOL; (*STN 1 ULTRASONIC FREQ ON/OFF (-16U1) *)
	WY10206_26 AT  %MX10224.26 : BOOL; (*STN 1 ULTRASONIC FREQ ON/OFF (-16U1) *)
	WY10206_27 AT  %MX10224.27 : BOOL; (*STN 1 ULTRASONIC FREQ ON/OFF (-16U1) *)
	WY10206_28 AT  %MX10224.28 : BOOL; (*STN 1 ULTRASONIC FREQ ON/OFF (-16U1) *)
	WY10206_29 AT  %MX10224.29 : BOOL; (*STN 1 ULTRASONIC FREQ ON/OFF (-16U1) *)
	WY10206_30 AT  %MX10224.30 : BOOL; (*STN 1 ULTRASONIC FREQ ON/OFF (-16U1) *)
	WY10206_31 AT  %MX10224.31 : BOOL; (*STN 1 ULTRASONIC FREQ ON/OFF (-16U1) *)

	WY10207_00 AT  %MX10228.0 : BOOL; (*STN 2 ULTRASONIC FREQ ON/OFF (-17U1) *)
	WY10207_01 AT  %MX10228.1 : BOOL; (*STN 2 ULTRASONIC FREQ ON/OFF (-17U1) *)
	WY10207_02 AT  %MX10228.2 : BOOL; (*STN 2 ULTRASONIC FREQ ON/OFF (-17U1) *)
	WY10207_03 AT  %MX10228.3 : BOOL; (*STN 2 ULTRASONIC FREQ ON/OFF (-17U1) *)
	WY10207_04 AT  %MX10228.4 : BOOL; (*STN 2 ULTRASONIC FREQ ON/OFF (-17U1) *)
	WY10207_05 AT  %MX10228.5 : BOOL; (*STN 2 ULTRASONIC FREQ ON/OFF (-17U1) *)
	WY10207_06 AT  %MX10228.6 : BOOL; (*STN 2 ULTRASONIC FREQ ON/OFF (-17U1) *)
	WY10207_07 AT  %MX10228.7 : BOOL; (*STN 2 ULTRASONIC FREQ ON/OFF (-17U1) *)
	WY10207_08 AT  %MX10228.8 : BOOL; (*STN 2 ULTRASONIC FREQ ON/OFF (-17U1) *)
	WY10207_09 AT  %MX10228.9 : BOOL; (*STN 2 ULTRASONIC FREQ ON/OFF (-17U1) *)
	WY10207_10 AT  %MX10228.10 : BOOL; (*STN 2 ULTRASONIC FREQ ON/OFF (-17U1) *)
	WY10207_11 AT  %MX10228.11 : BOOL; (*STN 2 ULTRASONIC FREQ ON/OFF (-17U1) *)
	WY10207_12 AT  %MX10228.12 : BOOL; (*STN 2 ULTRASONIC FREQ ON/OFF (-17U1) *)
	WY10207_13 AT  %MX10228.13 : BOOL; (*STN 2 ULTRASONIC FREQ ON/OFF (-17U1) *)
	WY10207_14 AT  %MX10228.14 : BOOL; (*STN 2 ULTRASONIC FREQ ON/OFF (-17U1) *)
	WY10207_15 AT  %MX10228.15 : BOOL; (*STN 2 ULTRASONIC FREQ ON/OFF (-17U1) *)
	WY10207_16 AT  %MX10228.16 : BOOL; (*STN 2 ULTRASONIC FREQ ON/OFF (-17U1) *)
	WY10207_17 AT  %MX10228.17 : BOOL; (*STN 2 ULTRASONIC FREQ ON/OFF (-17U1) *)
	WY10207_18 AT  %MX10228.18 : BOOL; (*STN 2 ULTRASONIC FREQ ON/OFF (-17U1) *)
	WY10207_19 AT  %MX10228.19 : BOOL; (*STN 2 ULTRASONIC FREQ ON/OFF (-17U1) *)
	WY10207_20 AT  %MX10228.20 : BOOL; (*STN 2 ULTRASONIC FREQ ON/OFF (-17U1) *)
	WY10207_21 AT  %MX10228.21 : BOOL; (*STN 2 ULTRASONIC FREQ ON/OFF (-17U1) *)
	WY10207_22 AT  %MX10228.22 : BOOL; (*STN 2 ULTRASONIC FREQ ON/OFF (-17U1) *)
	WY10207_23 AT  %MX10228.23 : BOOL; (*STN 2 ULTRASONIC FREQ ON/OFF (-17U1) *)
	WY10207_24 AT  %MX10228.24 : BOOL; (*STN 2 ULTRASONIC FREQ ON/OFF (-17U1) *)
	WY10207_25 AT  %MX10228.25 : BOOL; (*STN 2 ULTRASONIC FREQ ON/OFF (-17U1) *)
	WY10207_26 AT  %MX10228.26 : BOOL; (*STN 2 ULTRASONIC FREQ ON/OFF (-17U1) *)
	WY10207_27 AT  %MX10228.27 : BOOL; (*STN 2 ULTRASONIC FREQ ON/OFF (-17U1) *)
	WY10207_28 AT  %MX10228.28 : BOOL; (*STN 2 ULTRASONIC FREQ ON/OFF (-17U1) *)
	WY10207_29 AT  %MX10228.29 : BOOL; (*STN 2 ULTRASONIC FREQ ON/OFF (-17U1) *)
	WY10207_30 AT  %MX10228.30 : BOOL; (*STN 2 ULTRASONIC FREQ ON/OFF (-17U1) *)
	WY10207_31 AT  %MX10228.31 : BOOL; (*STN 2 ULTRASONIC FREQ ON/OFF (-17U1) *)

	WY10208_00 AT  %MX10232.0 : BOOL; (*STN 3 ULTRASONIC FREQ ON/OFF (-18U1) *)
	WY10208_01 AT  %MX10232.1 : BOOL; (*STN 3 ULTRASONIC FREQ ON/OFF (-18U1) *)
	WY10208_02 AT  %MX10232.2 : BOOL; (*STN 3 ULTRASONIC FREQ ON/OFF (-18U1) *)
	WY10208_03 AT  %MX10232.3 : BOOL; (*STN 3 ULTRASONIC FREQ ON/OFF (-18U1) *)
	WY10208_04 AT  %MX10232.4 : BOOL; (*STN 3 ULTRASONIC FREQ ON/OFF (-18U1) *)
	WY10208_05 AT  %MX10232.5 : BOOL; (*STN 3 ULTRASONIC FREQ ON/OFF (-18U1) *)
	WY10208_06 AT  %MX10232.6 : BOOL; (*STN 3 ULTRASONIC FREQ ON/OFF (-18U1) *)
	WY10208_07 AT  %MX10232.7 : BOOL; (*STN 3 ULTRASONIC FREQ ON/OFF (-18U1) *)
	WY10208_08 AT  %MX10232.8 : BOOL; (*STN 3 ULTRASONIC FREQ ON/OFF (-18U1) *)
	WY10208_09 AT  %MX10232.9 : BOOL; (*STN 3 ULTRASONIC FREQ ON/OFF (-18U1) *)
	WY10208_10 AT  %MX10232.10 : BOOL; (*STN 3 ULTRASONIC FREQ ON/OFF (-18U1) *)
	WY10208_11 AT  %MX10232.11 : BOOL; (*STN 3 ULTRASONIC FREQ ON/OFF (-18U1) *)
	WY10208_12 AT  %MX10232.12 : BOOL; (*STN 3 ULTRASONIC FREQ ON/OFF (-18U1) *)
	WY10208_13 AT  %MX10232.13 : BOOL; (*STN 3 ULTRASONIC FREQ ON/OFF (-18U1) *)
	WY10208_14 AT  %MX10232.14 : BOOL; (*STN 3 ULTRASONIC FREQ ON/OFF (-18U1) *)
	WY10208_15 AT  %MX10232.15 : BOOL; (*STN 3 ULTRASONIC FREQ ON/OFF (-18U1) *)
	WY10208_16 AT  %MX10232.16 : BOOL; (*STN 3 ULTRASONIC FREQ ON/OFF (-18U1) *)
	WY10208_17 AT  %MX10232.17 : BOOL; (*STN 3 ULTRASONIC FREQ ON/OFF (-18U1) *)
	WY10208_18 AT  %MX10232.18 : BOOL; (*STN 3 ULTRASONIC FREQ ON/OFF (-18U1) *)
	WY10208_19 AT  %MX10232.19 : BOOL; (*STN 3 ULTRASONIC FREQ ON/OFF (-18U1) *)
	WY10208_20 AT  %MX10232.20 : BOOL; (*STN 3 ULTRASONIC FREQ ON/OFF (-18U1) *)
	WY10208_21 AT  %MX10232.21 : BOOL; (*STN 3 ULTRASONIC FREQ ON/OFF (-18U1) *)
	WY10208_22 AT  %MX10232.22 : BOOL; (*STN 3 ULTRASONIC FREQ ON/OFF (-18U1) *)
	WY10208_23 AT  %MX10232.23 : BOOL; (*STN 3 ULTRASONIC FREQ ON/OFF (-18U1) *)
	WY10208_24 AT  %MX10232.24 : BOOL; (*STN 3 ULTRASONIC FREQ ON/OFF (-18U1) *)
	WY10208_25 AT  %MX10232.25 : BOOL; (*STN 3 ULTRASONIC FREQ ON/OFF (-18U1) *)
	WY10208_26 AT  %MX10232.26 : BOOL; (*STN 3 ULTRASONIC FREQ ON/OFF (-18U1) *)
	WY10208_27 AT  %MX10232.27 : BOOL; (*STN 3 ULTRASONIC FREQ ON/OFF (-18U1) *)
	WY10208_28 AT  %MX10232.28 : BOOL; (*STN 3 ULTRASONIC FREQ ON/OFF (-18U1) *)
	WY10208_29 AT  %MX10232.29 : BOOL; (*STN 3 ULTRASONIC FREQ ON/OFF (-18U1) *)
	WY10208_30 AT  %MX10232.30 : BOOL; (*STN 3 ULTRASONIC FREQ ON/OFF (-18U1) *)
	WY10208_31 AT  %MX10232.31 : BOOL; (*STN 3 ULTRASONIC FREQ ON/OFF (-18U1) *)

